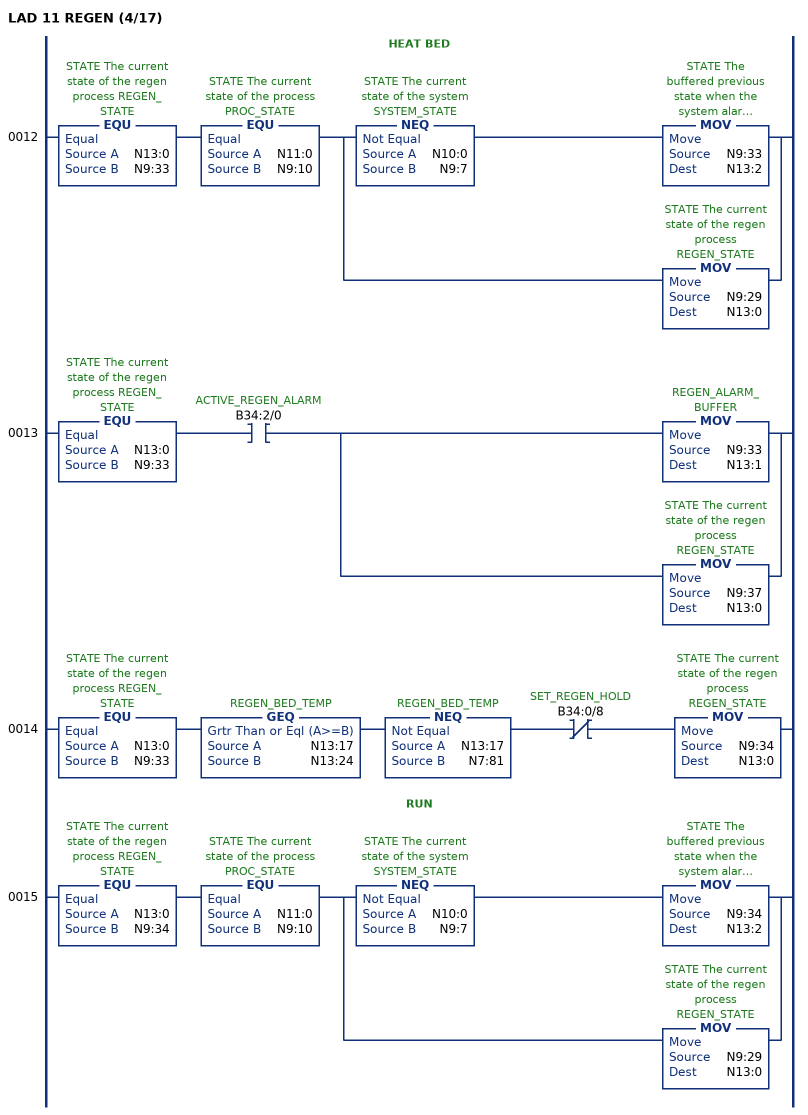
% Rung: 12 %
% TITLE: HEAT BED %
SOR EQU N13:0 N9:33 EQU N11:0 N9:10 BST NEQ N10:0 N9:7 MOV N9:33 N13:2 NXB MOV N9:29 N13:0 BND EOR
%   N13:0  REGEN_STATE  "STATE The current state of the regen process" %
%   N9:33  REGEN_HEAT_BED  "STATE Regen Heat wall" %
%   N11:0  PROC_STATE  "STATE The current state of the process" %
%   N9:10  PROC_STANDBY  "STATE Process Standby" %
%   N10:0  SYSTEM_STATE  "STATE The current state of the system" %
%   N9:7  SYSTEM_COLD_START %
%   N13:2  REGEN_SYSTEM_BUFFER  "STATE The buffered previous state when the system alarm occured" %
%   N9:29  REGEN_IDLE %
% Rung: 13 %
SOR EQU N13:0 N9:33 XIC B34:2/0 BST MOV N9:33 N13:1 NXB MOV N9:37 N13:0 BND EOR
%   N13:0  REGEN_STATE  "STATE The current state of the regen process" %
%   N9:33  REGEN_HEAT_BED  "STATE Regen Heat wall" %
%   B34:2/0  ACTIVE_REGEN_ALARM %
%   N13:1  REGEN_ALARM_BUFFER %
%   N9:37  REGEN_ALARM  "STATE Regen Alarm" %
% Rung: 14 %
SOR EQU N13:0 N9:33 GEQ N13:17 N13:24 NEQ N13:17 N7:81 XIO B34:0/8 MOV N9:34 N13:0 EOR
%   N13:0  REGEN_STATE  "STATE The current state of the regen process" %
%   N9:33  REGEN_HEAT_BED  "STATE Regen Heat wall" %
%   N13:17  REGEN_BED_TEMP %
%   N13:24  ADS_BED_TEMP_HIGH  "CONFIG The temp at which the regen process may continue" %
%   N7:81  TC_OPEN_SP  "CONFIG The value read by an open TC input" %
%   B34:0/8  SET_REGEN_HOLD %
%   N9:34  REGEN_RUN  "STATE Regen Running" %
% Rung: 15 %
% TITLE: RUN %
SOR EQU N13:0 N9:34 EQU N11:0 N9:10 BST NEQ N10:0 N9:7 MOV N9:34 N13:2 NXB MOV N9:29 N13:0 BND EOR
%   N13:0  REGEN_STATE  "STATE The current state of the regen process" %
%   N9:34  REGEN_RUN  "STATE Regen Running" %
%   N11:0  PROC_STATE  "STATE The current state of the process" %
%   N9:10  PROC_STANDBY  "STATE Process Standby" %
%   N10:0  SYSTEM_STATE  "STATE The current state of the system" %
%   N9:7  SYSTEM_COLD_START %
%   N13:2  REGEN_SYSTEM_BUFFER  "STATE The buffered previous state when the system alarm occured" %
%   N9:29  REGEN_IDLE %

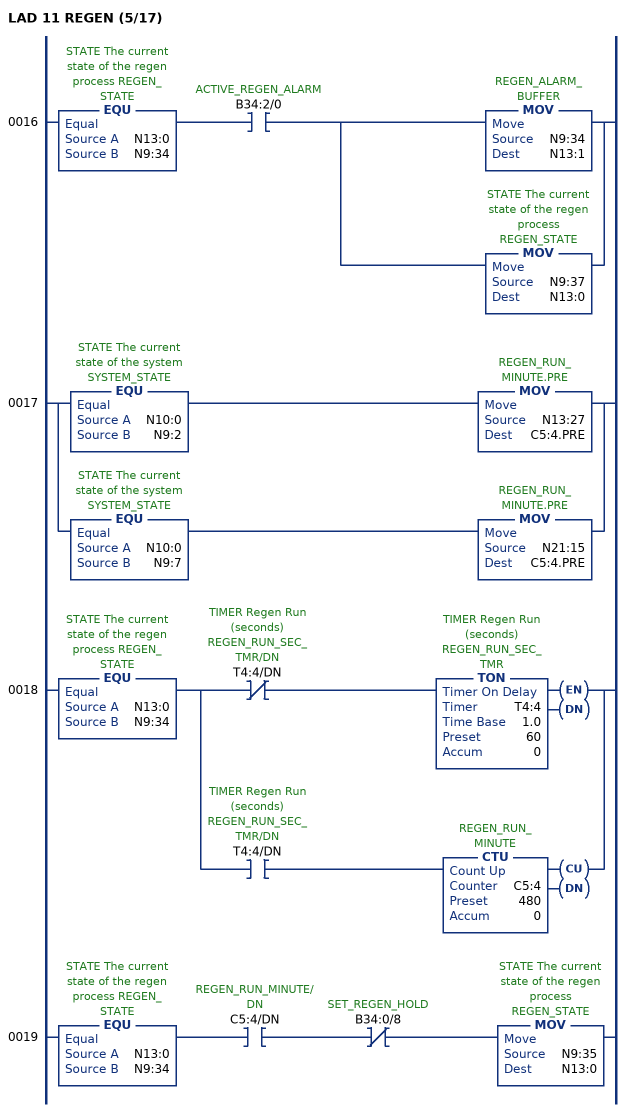
% Rung: 16 %
SOR EQU N13:0 N9:34 XIC B34:2/0 BST MOV N9:34 N13:1 NXB MOV N9:37 N13:0 BND EOR
%   N13:0  REGEN_STATE  "STATE The current state of the regen process" %
%   N9:34  REGEN_RUN  "STATE Regen Running" %
%   B34:2/0  ACTIVE_REGEN_ALARM %
%   N13:1  REGEN_ALARM_BUFFER %
%   N9:37  REGEN_ALARM  "STATE Regen Alarm" %
% Rung: 17 %
SOR BST EQU N10:0 N9:2 MOV N13:27 C5:4.PRE NXB EQU N10:0 N9:7 MOV N21:15 C5:4.PRE BND EOR
%   N10:0  SYSTEM_STATE  "STATE The current state of the system" %
%   N9:2  SYSTEM_PROCESS  "STATE System Process" %
%   N13:27  REGEN_RUN_TIME %
%   C5:4  REGEN_RUN_MINUTE %
%   N9:7  SYSTEM_COLD_START %
%   N21:15  START_REG_RUN_TIME %
% Rung: 18 %
SOR EQU N13:0 N9:34 BST XIO T4:4/DN TON T4:4 1.0 60 0 NXB XIC T4:4/DN CTU C5:4 480 0 BND EOR
%   N13:0  REGEN_STATE  "STATE The current state of the regen process" %
%   N9:34  REGEN_RUN  "STATE Regen Running" %
%   T4:4  REGEN_RUN_SEC_TMR  "TIMER Regen Run (seconds)" %
%   C5:4  REGEN_RUN_MINUTE %
% Rung: 19 %
SOR EQU N13:0 N9:34 XIC C5:4/DN XIO B34:0/8 MOV N9:35 N13:0 EOR
%   N13:0  REGEN_STATE  "STATE The current state of the regen process" %
%   N9:34  REGEN_RUN  "STATE Regen Running" %
%   C5:4  REGEN_RUN_MINUTE %
%   B34:0/8  SET_REGEN_HOLD %
%   N9:35  REGEN_COOL_WALL  "STATE Regen Cool wall" %

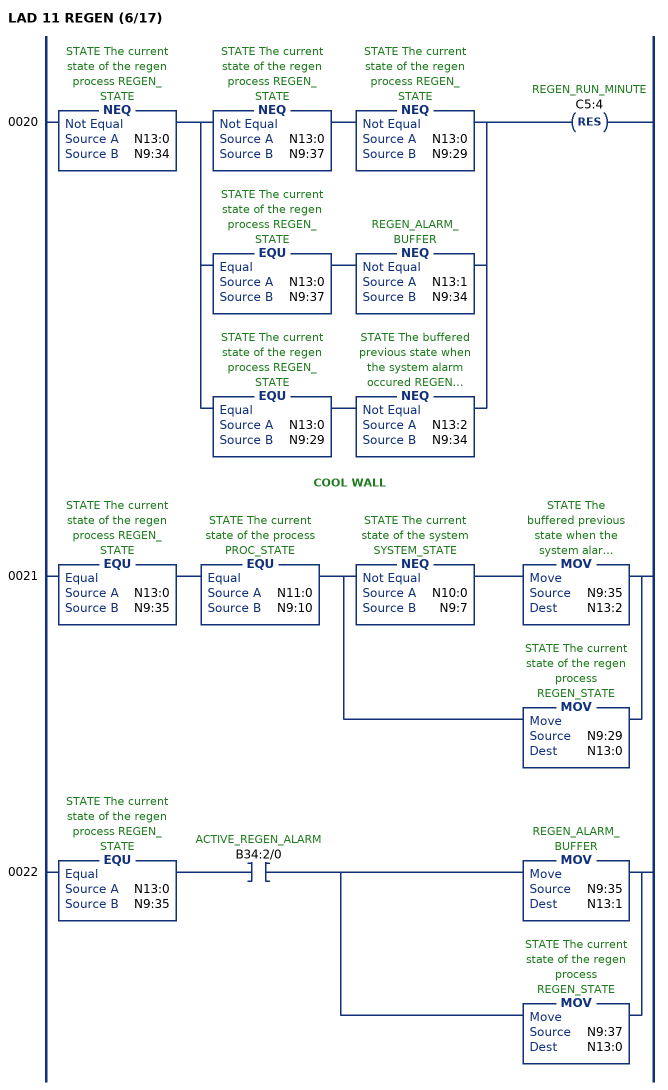
% Rung: 20 %
SOR NEQ N13:0 N9:34 BST NEQ N13:0 N9:37 NEQ N13:0 N9:29 NXB EQU N13:0 N9:37 NEQ N13:1 N9:34 NXB EQU N13:0 N9:29 NEQ N13:2 N9:34 BND RES C5:4 EOR
%   N13:0  REGEN_STATE  "STATE The current state of the regen process" %
%   N9:34  REGEN_RUN  "STATE Regen Running" %
%   N9:37  REGEN_ALARM  "STATE Regen Alarm" %
%   N9:29  REGEN_IDLE %
%   N13:1  REGEN_ALARM_BUFFER %
%   N13:2  REGEN_SYSTEM_BUFFER  "STATE The buffered previous state when the system alarm occured" %
%   C5:4  REGEN_RUN_MINUTE %
% Rung: 21 %
% TITLE: COOL WALL %
SOR EQU N13:0 N9:35 EQU N11:0 N9:10 BST NEQ N10:0 N9:7 MOV N9:35 N13:2 NXB MOV N9:29 N13:0 BND EOR
%   N13:0  REGEN_STATE  "STATE The current state of the regen process" %
%   N9:35  REGEN_COOL_WALL  "STATE Regen Cool wall" %
%   N11:0  PROC_STATE  "STATE The current state of the process" %
%   N9:10  PROC_STANDBY  "STATE Process Standby" %
%   N10:0  SYSTEM_STATE  "STATE The current state of the system" %
%   N9:7  SYSTEM_COLD_START %
%   N13:2  REGEN_SYSTEM_BUFFER  "STATE The buffered previous state when the system alarm occured" %
%   N9:29  REGEN_IDLE %
% Rung: 22 %
SOR EQU N13:0 N9:35 XIC B34:2/0 BST MOV N9:35 N13:1 NXB MOV N9:37 N13:0 BND EOR
%   N13:0  REGEN_STATE  "STATE The current state of the regen process" %
%   N9:35  REGEN_COOL_WALL  "STATE Regen Cool wall" %
%   B34:2/0  ACTIVE_REGEN_ALARM %
%   N13:1  REGEN_ALARM_BUFFER %
%   N9:37  REGEN_ALARM  "STATE Regen Alarm" %

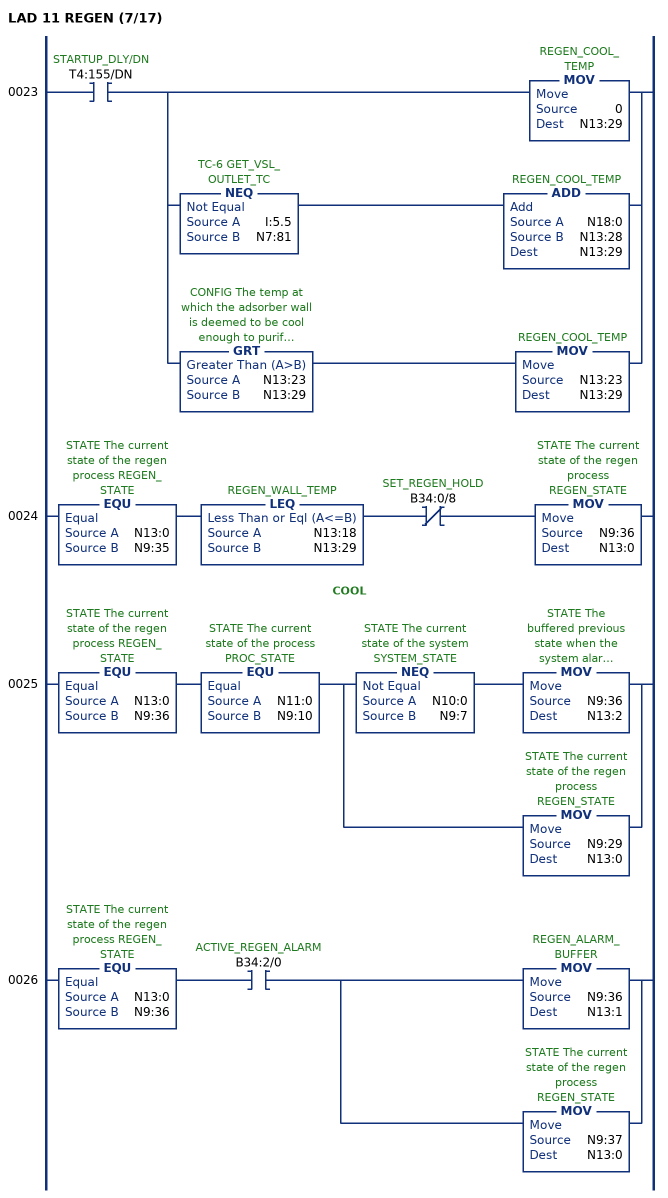
% Rung: 23 %
SOR XIC T4:155/DN BST MOV 0 N13:29 NXB NEQ I:5.5 N7:81 ADD N18:0 N13:28 N13:29 NXB GRT N13:23 N13:29 MOV N13:23 N13:29 BND EOR
%   T4:155  STARTUP_DLY %
%   N13:29  REGEN_COOL_TEMP %
%   I:5.5  GET_VSL_OUTLET_TC  "TC-6" %
%   N7:81  TC_OPEN_SP  "CONFIG The value read by an open TC input" %
%   N18:0  GET_VSL_OUT_GAS_TEMP %
%   N13:28  REGEN_COOL_DIFF %
%   N13:23  ADS_WALL_TEMP_COOL  "CONFIG The temp at which the adsorber wall is deemed to be cool enough to purify" %
% Rung: 24 %
SOR EQU N13:0 N9:35 LEQ N13:18 N13:29 XIO B34:0/8 MOV N9:36 N13:0 EOR
%   N13:0  REGEN_STATE  "STATE The current state of the regen process" %
%   N9:35  REGEN_COOL_WALL  "STATE Regen Cool wall" %
%   N13:18  REGEN_WALL_TEMP %
%   N13:29  REGEN_COOL_TEMP %
%   B34:0/8  SET_REGEN_HOLD %
%   N9:36  REGEN_COOL  "STATE Regen Cool" %
% Rung: 25 %
% TITLE: COOL %
SOR EQU N13:0 N9:36 EQU N11:0 N9:10 BST NEQ N10:0 N9:7 MOV N9:36 N13:2 NXB MOV N9:29 N13:0 BND EOR
%   N13:0  REGEN_STATE  "STATE The current state of the regen process" %
%   N9:36  REGEN_COOL  "STATE Regen Cool" %
%   N11:0  PROC_STATE  "STATE The current state of the process" %
%   N9:10  PROC_STANDBY  "STATE Process Standby" %
%   N10:0  SYSTEM_STATE  "STATE The current state of the system" %
%   N9:7  SYSTEM_COLD_START %
%   N13:2  REGEN_SYSTEM_BUFFER  "STATE The buffered previous state when the system alarm occured" %
%   N9:29  REGEN_IDLE %
% Rung: 26 %
SOR EQU N13:0 N9:36 XIC B34:2/0 BST MOV N9:36 N13:1 NXB MOV N9:37 N13:0 BND EOR
%   N13:0  REGEN_STATE  "STATE The current state of the regen process" %
%   N9:36  REGEN_COOL  "STATE Regen Cool" %
%   B34:2/0  ACTIVE_REGEN_ALARM %
%   N13:1  REGEN_ALARM_BUFFER %
%   N9:37  REGEN_ALARM  "STATE Regen Alarm" %

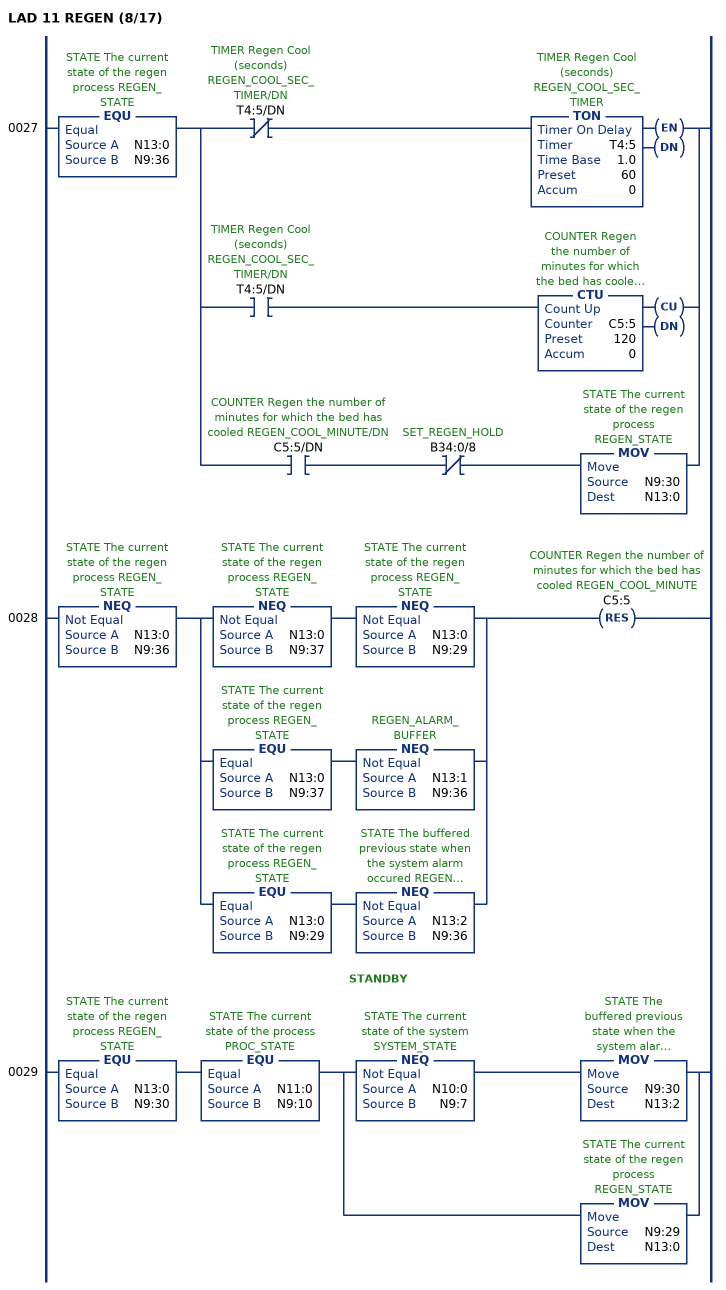
% Rung: 27 %
SOR EQU N13:0 N9:36 BST XIO T4:5/DN TON T4:5 1.0 60 0 NXB XIC T4:5/DN CTU C5:5 120 0 NXB XIC C5:5/DN XIO B34:0/8 MOV N9:30 N13:0 BND EOR
%   N13:0  REGEN_STATE  "STATE The current state of the regen process" %
%   N9:36  REGEN_COOL  "STATE Regen Cool" %
%   T4:5  REGEN_COOL_SEC_TIMER  "TIMER Regen Cool (seconds)" %
%   C5:5  REGEN_COOL_MINUTE  "COUNTER Regen the number of minutes for which the bed has cooled" %
%   B34:0/8  SET_REGEN_HOLD %
%   N9:30  REGEN_STANDBY  "STATE Regen Standby" %
% Rung: 28 %
SOR NEQ N13:0 N9:36 BST NEQ N13:0 N9:37 NEQ N13:0 N9:29 NXB EQU N13:0 N9:37 NEQ N13:1 N9:36 NXB EQU N13:0 N9:29 NEQ N13:2 N9:36 BND RES C5:5 EOR
%   N13:0  REGEN_STATE  "STATE The current state of the regen process" %
%   N9:36  REGEN_COOL  "STATE Regen Cool" %
%   N9:37  REGEN_ALARM  "STATE Regen Alarm" %
%   N9:29  REGEN_IDLE %
%   N13:1  REGEN_ALARM_BUFFER %
%   N13:2  REGEN_SYSTEM_BUFFER  "STATE The buffered previous state when the system alarm occured" %
%   C5:5  REGEN_COOL_MINUTE  "COUNTER Regen the number of minutes for which the bed has cooled" %
% Rung: 29 %
% TITLE: STANDBY %
SOR EQU N13:0 N9:30 EQU N11:0 N9:10 BST NEQ N10:0 N9:7 MOV N9:30 N13:2 NXB MOV N9:29 N13:0 BND EOR
%   N13:0  REGEN_STATE  "STATE The current state of the regen process" %
%   N9:30  REGEN_STANDBY  "STATE Regen Standby" %
%   N11:0  PROC_STATE  "STATE The current state of the process" %
%   N9:10  PROC_STANDBY  "STATE Process Standby" %
%   N10:0  SYSTEM_STATE  "STATE The current state of the system" %
%   N9:7  SYSTEM_COLD_START %
%   N13:2  REGEN_SYSTEM_BUFFER  "STATE The buffered previous state when the system alarm occured" %
%   N9:29  REGEN_IDLE %

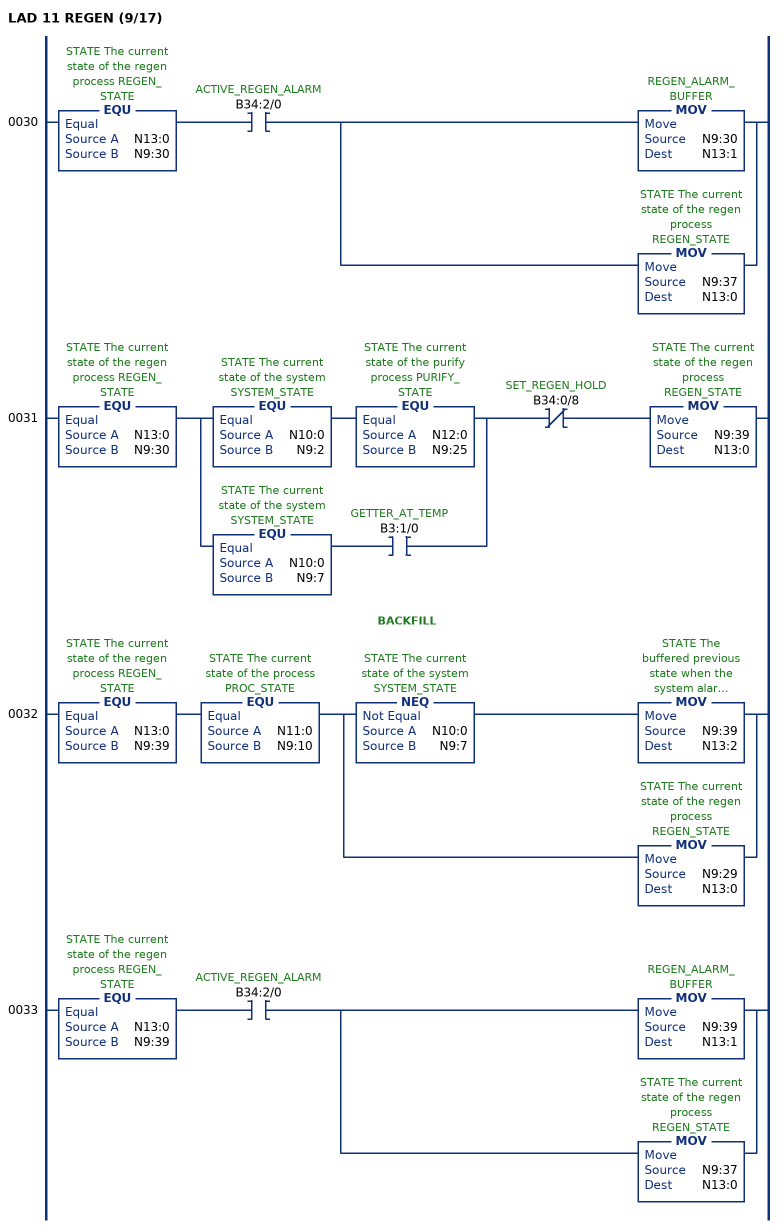
% Rung: 30 %
SOR EQU N13:0 N9:30 XIC B34:2/0 BST MOV N9:30 N13:1 NXB MOV N9:37 N13:0 BND EOR
%   N13:0  REGEN_STATE  "STATE The current state of the regen process" %
%   N9:30  REGEN_STANDBY  "STATE Regen Standby" %
%   B34:2/0  ACTIVE_REGEN_ALARM %
%   N13:1  REGEN_ALARM_BUFFER %
%   N9:37  REGEN_ALARM  "STATE Regen Alarm" %
% Rung: 31 %
SOR EQU N13:0 N9:30 BST EQU N10:0 N9:2 EQU N12:0 N9:25 NXB EQU N10:0 N9:7 XIC B3:1/0 BND XIO B34:0/8 MOV N9:39 N13:0 EOR
%   N13:0  REGEN_STATE  "STATE The current state of the regen process" %
%   N9:30  REGEN_STANDBY  "STATE Regen Standby" %
%   N10:0  SYSTEM_STATE  "STATE The current state of the system" %
%   N9:2  SYSTEM_PROCESS  "STATE System Process" %
%   N12:0  PURIFY_STATE  "STATE The current state of the purify process" %
%   N9:25  PURIFY_DONE %
%   N9:7  SYSTEM_COLD_START %
%   B3:1/0  GETTER_AT_TEMP %
%   B34:0/8  SET_REGEN_HOLD %
%   N9:39  REGEN_BACKFILL %
% Rung: 32 %
% TITLE: BACKFILL %
SOR EQU N13:0 N9:39 EQU N11:0 N9:10 BST NEQ N10:0 N9:7 MOV N9:39 N13:2 NXB MOV N9:29 N13:0 BND EOR
%   N13:0  REGEN_STATE  "STATE The current state of the regen process" %
%   N9:39  REGEN_BACKFILL %
%   N11:0  PROC_STATE  "STATE The current state of the process" %
%   N9:10  PROC_STANDBY  "STATE Process Standby" %
%   N10:0  SYSTEM_STATE  "STATE The current state of the system" %
%   N9:7  SYSTEM_COLD_START %
%   N13:2  REGEN_SYSTEM_BUFFER  "STATE The buffered previous state when the system alarm occured" %
%   N9:29  REGEN_IDLE %
% Rung: 33 %
SOR EQU N13:0 N9:39 XIC B34:2/0 BST MOV N9:39 N13:1 NXB MOV N9:37 N13:0 BND EOR
%   N13:0  REGEN_STATE  "STATE The current state of the regen process" %
%   N9:39  REGEN_BACKFILL %
%   B34:2/0  ACTIVE_REGEN_ALARM %
%   N13:1  REGEN_ALARM_BUFFER %
%   N9:37  REGEN_ALARM  "STATE Regen Alarm" %

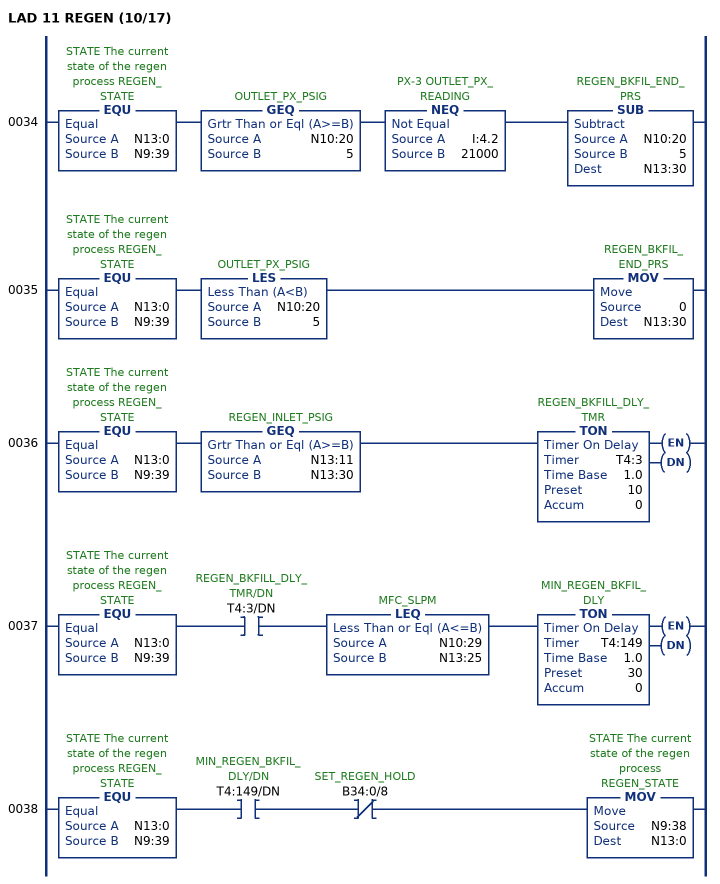
% Rung: 34 %
SOR EQU N13:0 N9:39 GEQ N10:20 5 NEQ I:4.2 21000 SUB N10:20 5 N13:30 EOR
%   N13:0  REGEN_STATE  "STATE The current state of the regen process" %
%   N9:39  REGEN_BACKFILL %
%   N10:20  OUTLET_PX_PSIG %
%   I:4.2  OUTLET_PX_READING  "PX-3" %
%   N13:30  REGEN_BKFIL_END_PRS %
% Rung: 35 %
SOR EQU N13:0 N9:39 LES N10:20 5 MOV 0 N13:30 EOR
%   N13:0  REGEN_STATE  "STATE The current state of the regen process" %
%   N9:39  REGEN_BACKFILL %
%   N10:20  OUTLET_PX_PSIG %
%   N13:30  REGEN_BKFIL_END_PRS %
% Rung: 36 %
SOR EQU N13:0 N9:39 GEQ N13:11 N13:30 TON T4:3 1.0 10 0 EOR
%   N13:0  REGEN_STATE  "STATE The current state of the regen process" %
%   N9:39  REGEN_BACKFILL %
%   N13:11  REGEN_INLET_PSIG %
%   N13:30  REGEN_BKFIL_END_PRS %
%   T4:3  REGEN_BKFILL_DLY_TMR %
% Rung: 37 %
SOR EQU N13:0 N9:39 XIC T4:3/DN LEQ N10:29 N13:25 TON T4:149 1.0 30 0 EOR
%   N13:0  REGEN_STATE  "STATE The current state of the regen process" %
%   N9:39  REGEN_BACKFILL %
%   T4:3  REGEN_BKFILL_DLY_TMR %
%   N10:29  MFC_SLPM %
%   N13:25  REGEN_BKFIL_END_FLOW %
%   T4:149  MIN_REGEN_BKFIL_DLY %
% Rung: 38 %
SOR EQU N13:0 N9:39 XIC T4:149/DN XIO B34:0/8 MOV N9:38 N13:0 EOR
%   N13:0  REGEN_STATE  "STATE The current state of the regen process" %
%   N9:39  REGEN_BACKFILL %
%   T4:149  MIN_REGEN_BKFIL_DLY %
%   B34:0/8  SET_REGEN_HOLD %
%   N9:38  REGEN_DONE %

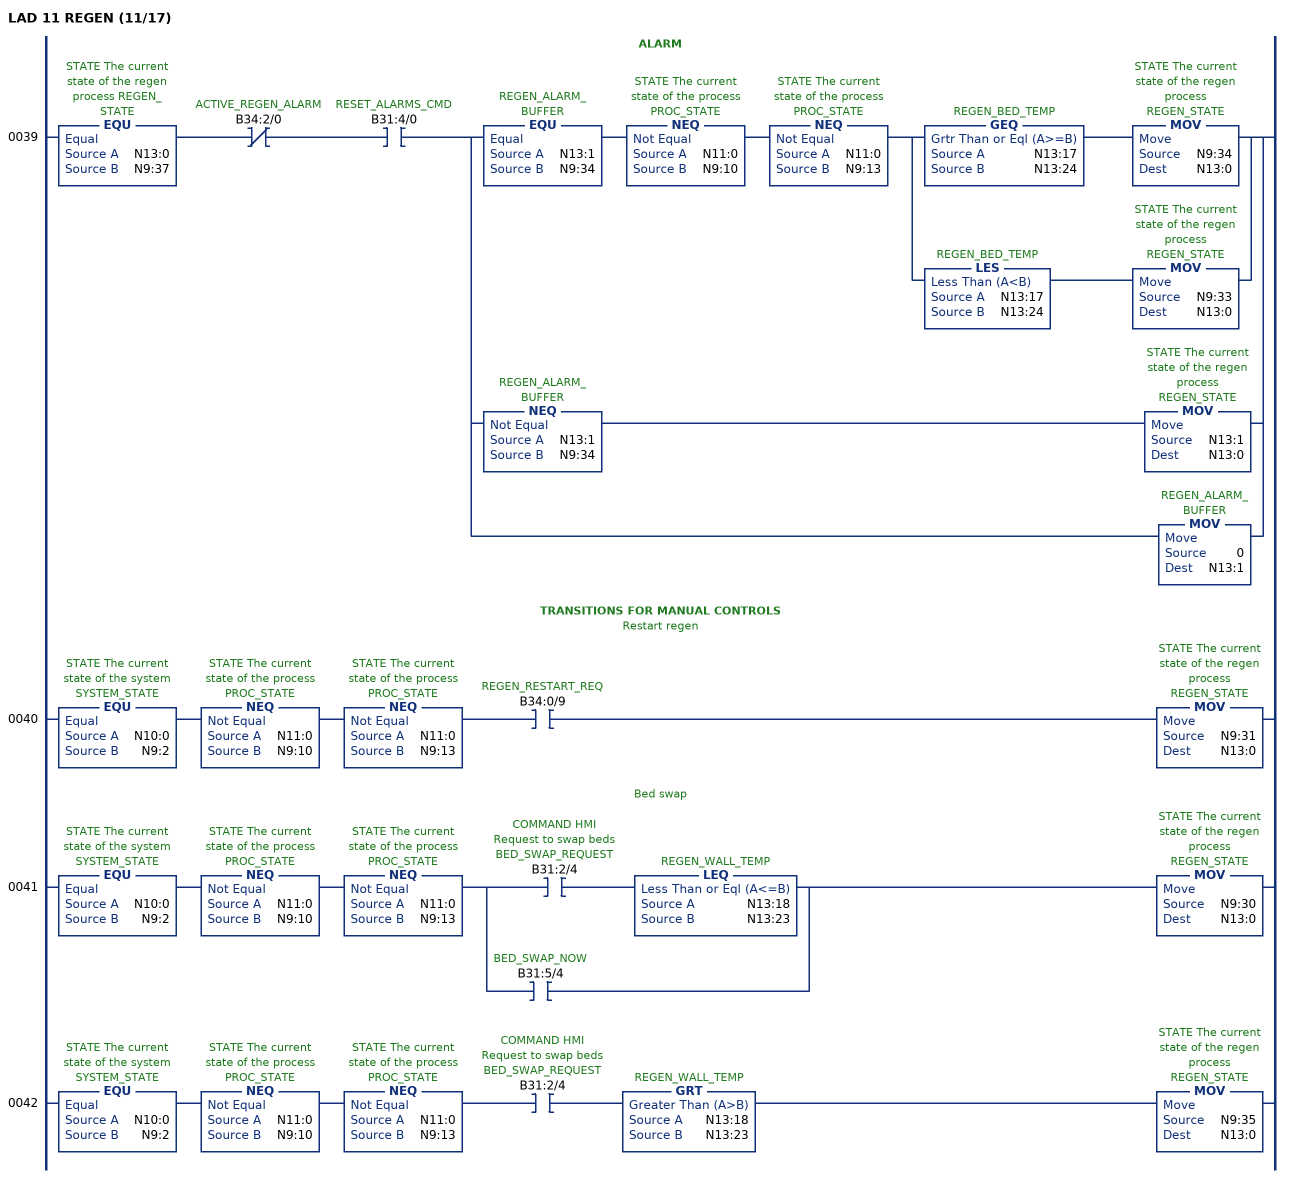
% Rung: 39 %
% TITLE: ALARM %
SOR EQU N13:0 N9:37 XIO B34:2/0 XIC B31:4/0 BST EQU N13:1 N9:34 NEQ N11:0 N9:10 NEQ N11:0 N9:13 BST GEQ N13:17 N13:24 MOV N9:34 N13:0 NXB LES N13:17 N13:24 MOV N9:33 N13:0 BND NXB NEQ N13:1 N9:34 MOV N13:1 N13:0 NXB MOV 0 N13:1 BND EOR
%   N13:0  REGEN_STATE  "STATE The current state of the regen process" %
%   N9:37  REGEN_ALARM  "STATE Regen Alarm" %
%   B34:2/0  ACTIVE_REGEN_ALARM %
%   B31:4/0  RESET_ALARMS_CMD %
%   N13:1  REGEN_ALARM_BUFFER %
%   N9:34  REGEN_RUN  "STATE Regen Running" %
%   N11:0  PROC_STATE  "STATE The current state of the process" %
%   N9:10  PROC_STANDBY  "STATE Process Standby" %
%   N9:13  PROC_OVERLAP  "STATE Process Purify Overlap" %
%   N13:17  REGEN_BED_TEMP %
%   N13:24  ADS_BED_TEMP_HIGH  "CONFIG The temp at which the regen process may continue" %
%   N9:33  REGEN_HEAT_BED  "STATE Regen Heat wall" %
% Rung: 40 %
% TITLE: TRANSITIONS FOR MANUAL CONTROLS %
% Restart regen %
SOR EQU N10:0 N9:2 NEQ N11:0 N9:10 NEQ N11:0 N9:13 XIC B34:0/9 MOV N9:31 N13:0 EOR
%   N10:0  SYSTEM_STATE  "STATE The current state of the system" %
%   N9:2  SYSTEM_PROCESS  "STATE System Process" %
%   N11:0  PROC_STATE  "STATE The current state of the process" %
%   N9:10  PROC_STANDBY  "STATE Process Standby" %
%   N9:13  PROC_OVERLAP  "STATE Process Purify Overlap" %
%   B34:0/9  REGEN_RESTART_REQ %
%   N9:31  REGEN_DELAY  "STATE Regen Delay" %
%   N13:0  REGEN_STATE  "STATE The current state of the regen process" %
% Rung: 41 %
% Bed swap %
SOR EQU N10:0 N9:2 NEQ N11:0 N9:10 NEQ N11:0 N9:13 BST XIC B31:2/4 LEQ N13:18 N13:23 NXB XIC B31:5/4 BND MOV N9:30 N13:0 EOR
%   N10:0  SYSTEM_STATE  "STATE The current state of the system" %
%   N9:2  SYSTEM_PROCESS  "STATE System Process" %
%   N11:0  PROC_STATE  "STATE The current state of the process" %
%   N9:10  PROC_STANDBY  "STATE Process Standby" %
%   N9:13  PROC_OVERLAP  "STATE Process Purify Overlap" %
%   B31:2/4  BED_SWAP_REQUEST  "COMMAND HMI Request to swap beds" %
%   N13:18  REGEN_WALL_TEMP %
%   N13:23  ADS_WALL_TEMP_COOL  "CONFIG The temp at which the adsorber wall is deemed to be cool enough to purify" %
%   B31:5/4  BED_SWAP_NOW %
%   N9:30  REGEN_STANDBY  "STATE Regen Standby" %
%   N13:0  REGEN_STATE  "STATE The current state of the regen process" %
% Rung: 42 %
SOR EQU N10:0 N9:2 NEQ N11:0 N9:10 NEQ N11:0 N9:13 XIC B31:2/4 GRT N13:18 N13:23 MOV N9:35 N13:0 EOR
%   N10:0  SYSTEM_STATE  "STATE The current state of the system" %
%   N9:2  SYSTEM_PROCESS  "STATE System Process" %
%   N11:0  PROC_STATE  "STATE The current state of the process" %
%   N9:10  PROC_STANDBY  "STATE Process Standby" %
%   N9:13  PROC_OVERLAP  "STATE Process Purify Overlap" %
%   B31:2/4  BED_SWAP_REQUEST  "COMMAND HMI Request to swap beds" %
%   N13:18  REGEN_WALL_TEMP %
%   N13:23  ADS_WALL_TEMP_COOL  "CONFIG The temp at which the adsorber wall is deemed to be cool enough to purify" %
%   N9:35  REGEN_COOL_WALL  "STATE Regen Cool wall" %
%   N13:0  REGEN_STATE  "STATE The current state of the regen process" %

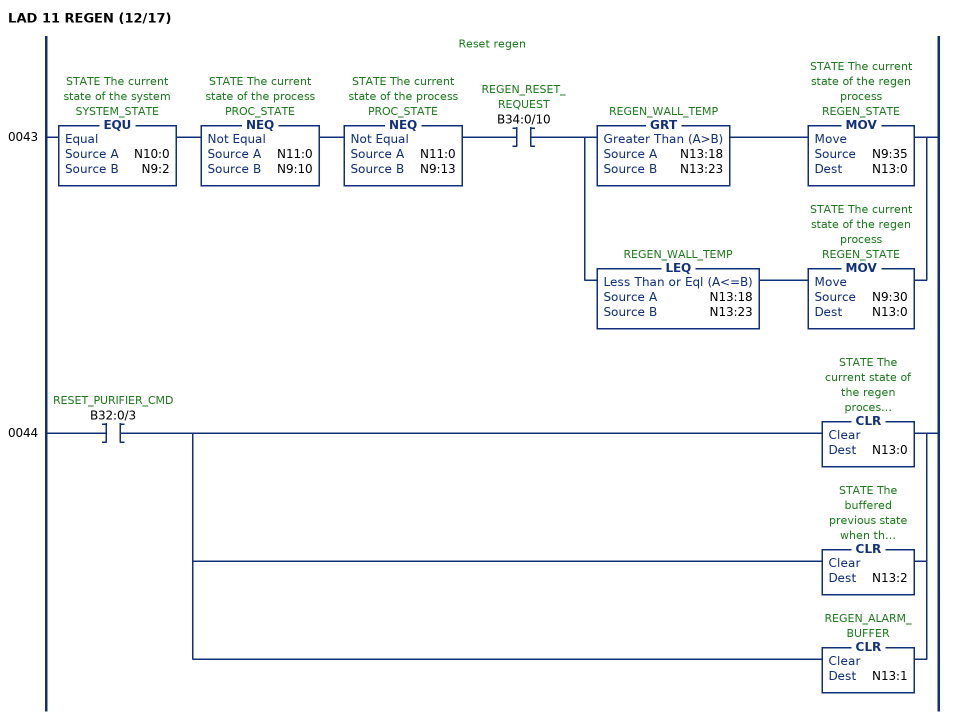
% Rung: 43 %
% Reset regen %
SOR EQU N10:0 N9:2 NEQ N11:0 N9:10 NEQ N11:0 N9:13 XIC B34:0/10 BST GRT N13:18 N13:23 MOV N9:35 N13:0 NXB LEQ N13:18 N13:23 MOV N9:30 N13:0 BND EOR
%   N10:0  SYSTEM_STATE  "STATE The current state of the system" %
%   N9:2  SYSTEM_PROCESS  "STATE System Process" %
%   N11:0  PROC_STATE  "STATE The current state of the process" %
%   N9:10  PROC_STANDBY  "STATE Process Standby" %
%   N9:13  PROC_OVERLAP  "STATE Process Purify Overlap" %
%   B34:0/10  REGEN_RESET_REQUEST %
%   N13:18  REGEN_WALL_TEMP %
%   N13:23  ADS_WALL_TEMP_COOL  "CONFIG The temp at which the adsorber wall is deemed to be cool enough to purify" %
%   N9:35  REGEN_COOL_WALL  "STATE Regen Cool wall" %
%   N13:0  REGEN_STATE  "STATE The current state of the regen process" %
%   N9:30  REGEN_STANDBY  "STATE Regen Standby" %
% Rung: 44 %
SOR XIC B32:0/3 BST CLR N13:0 NXB CLR N13:2 NXB CLR N13:1 BND EOR
%   B32:0/3  RESET_PURIFIER_CMD %
%   N13:0  REGEN_STATE  "STATE The current state of the regen process" %
%   N13:2  REGEN_SYSTEM_BUFFER  "STATE The buffered previous state when the system alarm occured" %
%   N13:1  REGEN_ALARM_BUFFER %

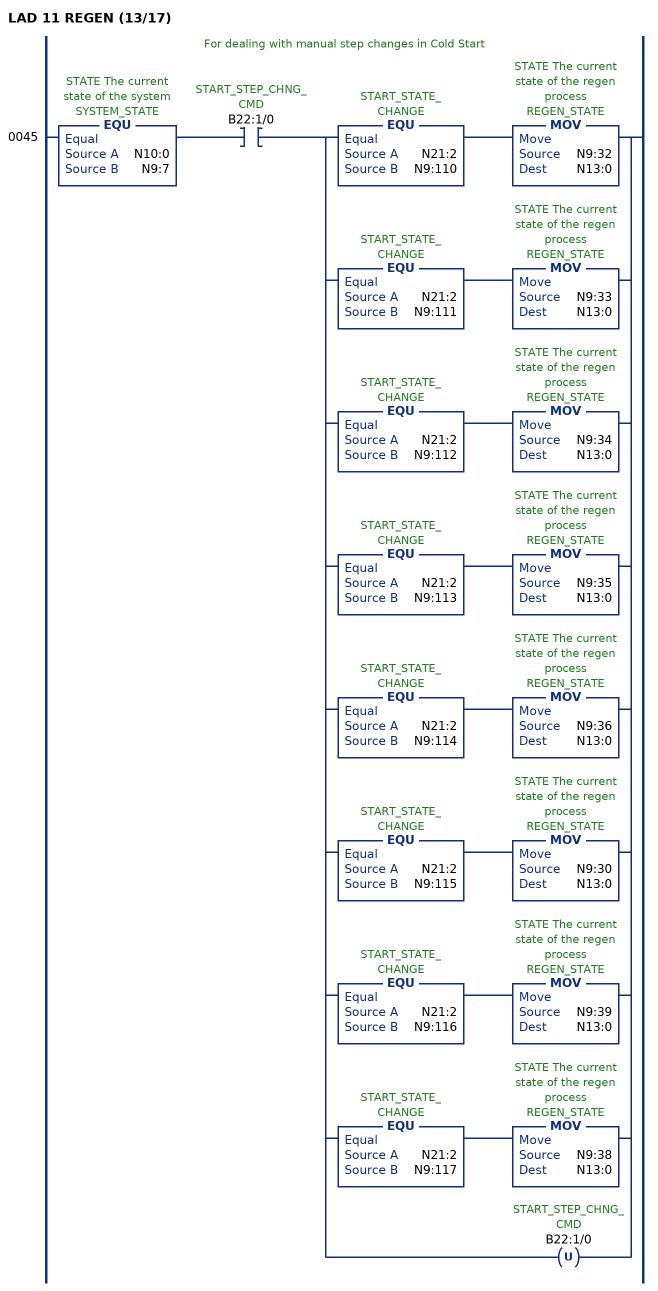
% Rung: 45 %
% For dealing with manual step changes in Cold Start %
SOR EQU N10:0 N9:7 XIC B22:1/0 BST EQU N21:2 N9:110 MOV N9:32 N13:0 NXB EQU N21:2 N9:111 MOV N9:33 N13:0 NXB EQU N21:2 N9:112 MOV N9:34 N13:0 NXB EQU N21:2 N9:113 MOV N9:35 N13:0 NXB EQU N21:2 N9:114 MOV N9:36 N13:0 NXB EQU N21:2 N9:115 MOV N9:30 N13:0 NXB EQU N21:2 N9:116 MOV N9:39 N13:0 NXB EQU N21:2 N9:117 MOV N9:38 N13:0 NXB OTU B22:1/0 BND EOR
%   N10:0  SYSTEM_STATE  "STATE The current state of the system" %
%   N9:7  SYSTEM_COLD_START %
%   B22:1/0  START_STEP_CHNG_CMD %
%   N21:2  START_STATE_CHANGE %
%   N9:110  START_REG_VENT %
%   N9:32  REGEN_VENT  "STATE Regen Vent" %
%   N13:0  REGEN_STATE  "STATE The current state of the regen process" %
%   N9:111  START_REG_HEAT %
%   N9:33  REGEN_HEAT_BED  "STATE Regen Heat wall" %
%   N9:112  START_REG_RUN %
%   N9:34  REGEN_RUN  "STATE Regen Running" %
%   N9:113  START_REG_COOL %
%   N9:35  REGEN_COOL_WALL  "STATE Regen Cool wall" %
%   N9:114  START_REG_TIMED_COOL %
%   N9:36  REGEN_COOL  "STATE Regen Cool" %
%   N9:115  START_REG_STANDBY %
%   N9:30  REGEN_STANDBY  "STATE Regen Standby" %
%   N9:116  START_REG_BACKFILL %
%   N9:39  REGEN_BACKFILL %
%   N9:117  START_REG_DONE %
%   N9:38  REGEN_DONE %

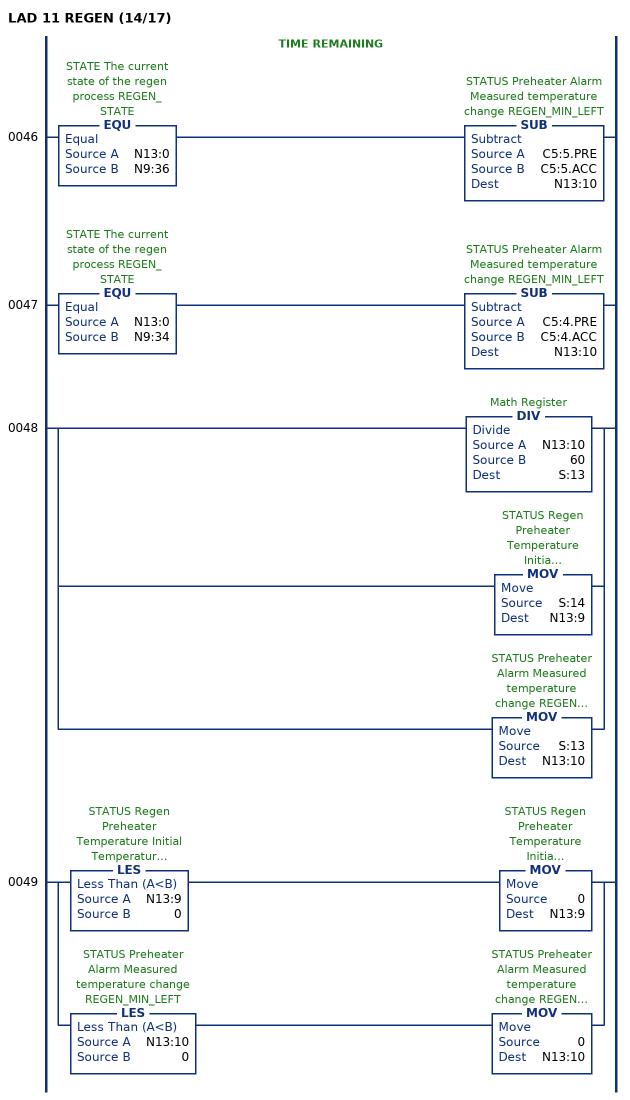
% Rung: 46 %
% TITLE: TIME REMAINING %
SOR EQU N13:0 N9:36 SUB C5:5.PRE C5:5.ACC N13:10 EOR
%   N13:0  REGEN_STATE  "STATE The current state of the regen process" %
%   N9:36  REGEN_COOL  "STATE Regen Cool" %
%   C5:5  REGEN_COOL_MINUTE  "COUNTER Regen the number of minutes for which the bed has cooled" %
%   N13:10  REGEN_MIN_LEFT  "STATUS Preheater Alarm Measured temperature change" %
% Rung: 47 %
SOR EQU N13:0 N9:34 SUB C5:4.PRE C5:4.ACC N13:10 EOR
%   N13:0  REGEN_STATE  "STATE The current state of the regen process" %
%   N9:34  REGEN_RUN  "STATE Regen Running" %
%   C5:4  REGEN_RUN_MINUTE %
%   N13:10  REGEN_MIN_LEFT  "STATUS Preheater Alarm Measured temperature change" %
% Rung: 48 %
SOR BST DIV N13:10 60 S:13 NXB MOV S:14 N13:9 NXB MOV S:13 N13:10 BND EOR
%   N13:10  REGEN_MIN_LEFT  "STATUS Preheater Alarm Measured temperature change" %
%   S:13  "Math Register" %
%   S:14  "Math Register" %
%   N13:9  REGEN_HRS_LEFT  "STATUS Regen Preheater Temperature Initial Temperature" %
% Rung: 49 %
SOR BST LES N13:9 0 MOV 0 N13:9 NXB LES N13:10 0 MOV 0 N13:10 BND EOR
%   N13:9  REGEN_HRS_LEFT  "STATUS Regen Preheater Temperature Initial Temperature" %
%   N13:10  REGEN_MIN_LEFT  "STATUS Preheater Alarm Measured temperature change" %

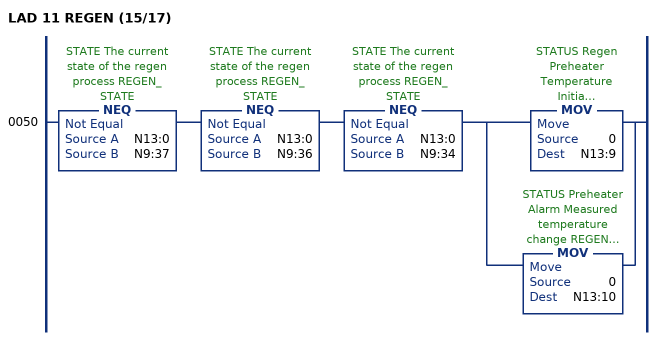
% Rung: 50 %
SOR NEQ N13:0 N9:37 NEQ N13:0 N9:36 NEQ N13:0 N9:34 BST MOV 0 N13:9 NXB MOV 0 N13:10 BND EOR
%   N13:0  REGEN_STATE  "STATE The current state of the regen process" %
%   N9:37  REGEN_ALARM  "STATE Regen Alarm" %
%   N9:36  REGEN_COOL  "STATE Regen Cool" %
%   N9:34  REGEN_RUN  "STATE Regen Running" %
%   N13:9  REGEN_HRS_LEFT  "STATUS Regen Preheater Temperature Initial Temperature" %
%   N13:10  REGEN_MIN_LEFT  "STATUS Preheater Alarm Measured temperature change" %

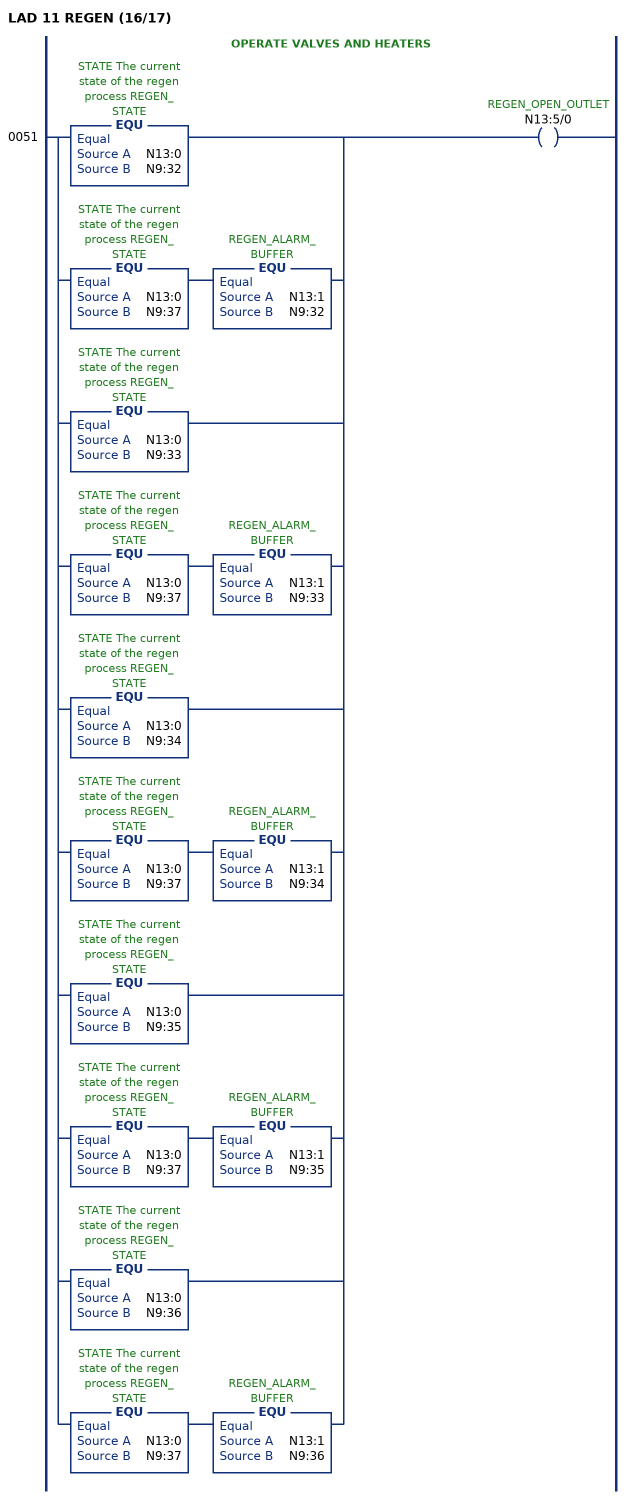
% Rung: 51 %
% TITLE: OPERATE VALVES AND HEATERS %
SOR BST EQU N13:0 N9:32 NXB EQU N13:0 N9:37 EQU N13:1 N9:32 NXB EQU N13:0 N9:33 NXB EQU N13:0 N9:37 EQU N13:1 N9:33 NXB EQU N13:0 N9:34 NXB EQU N13:0 N9:37 EQU N13:1 N9:34 NXB EQU N13:0 N9:35 NXB EQU N13:0 N9:37 EQU N13:1 N9:35 NXB EQU N13:0 N9:36 NXB EQU N13:0 N9:37 EQU N13:1 N9:36 BND OTE N13:5/0 EOR
%   N13:0  REGEN_STATE  "STATE The current state of the regen process" %
%   N9:32  REGEN_VENT  "STATE Regen Vent" %
%   N9:37  REGEN_ALARM  "STATE Regen Alarm" %
%   N13:1  REGEN_ALARM_BUFFER %
%   N9:33  REGEN_HEAT_BED  "STATE Regen Heat wall" %
%   N9:34  REGEN_RUN  "STATE Regen Running" %
%   N9:35  REGEN_COOL_WALL  "STATE Regen Cool wall" %
%   N9:36  REGEN_COOL  "STATE Regen Cool" %
%   N13:5/0  REGEN_OPEN_OUTLET %

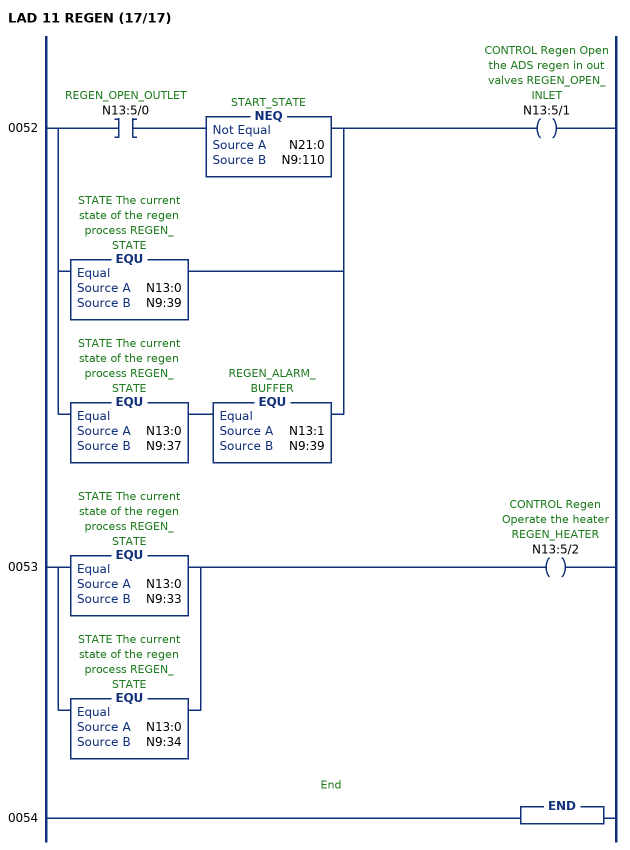
% Rung: 52 %
SOR BST XIC N13:5/0 NEQ N21:0 N9:110 NXB EQU N13:0 N9:39 NXB EQU N13:0 N9:37 EQU N13:1 N9:39 BND OTE N13:5/1 EOR
%   N13:5/0  REGEN_OPEN_OUTLET %
%   N21:0  START_STATE %
%   N9:110  START_REG_VENT %
%   N13:0  REGEN_STATE  "STATE The current state of the regen process" %
%   N9:39  REGEN_BACKFILL %
%   N9:37  REGEN_ALARM  "STATE Regen Alarm" %
%   N13:1  REGEN_ALARM_BUFFER %
%   N13:5/1  REGEN_OPEN_INLET  "CONTROL Regen Open the ADS regen in out valves" %
% Rung: 53 %
SOR BST EQU N13:0 N9:33 NXB EQU N13:0 N9:34 BND OTE N13:5/2 EOR
%   N13:0  REGEN_STATE  "STATE The current state of the regen process" %
%   N9:33  REGEN_HEAT_BED  "STATE Regen Heat wall" %
%   N9:34  REGEN_RUN  "STATE Regen Running" %
%   N13:5/2  REGEN_HEATER  "CONTROL Regen Operate the heater" %
% Rung: 54 %
% End %
SOR END EOR

LADDER 12 "REGEN_FLT"    % regen alarms and warnings %
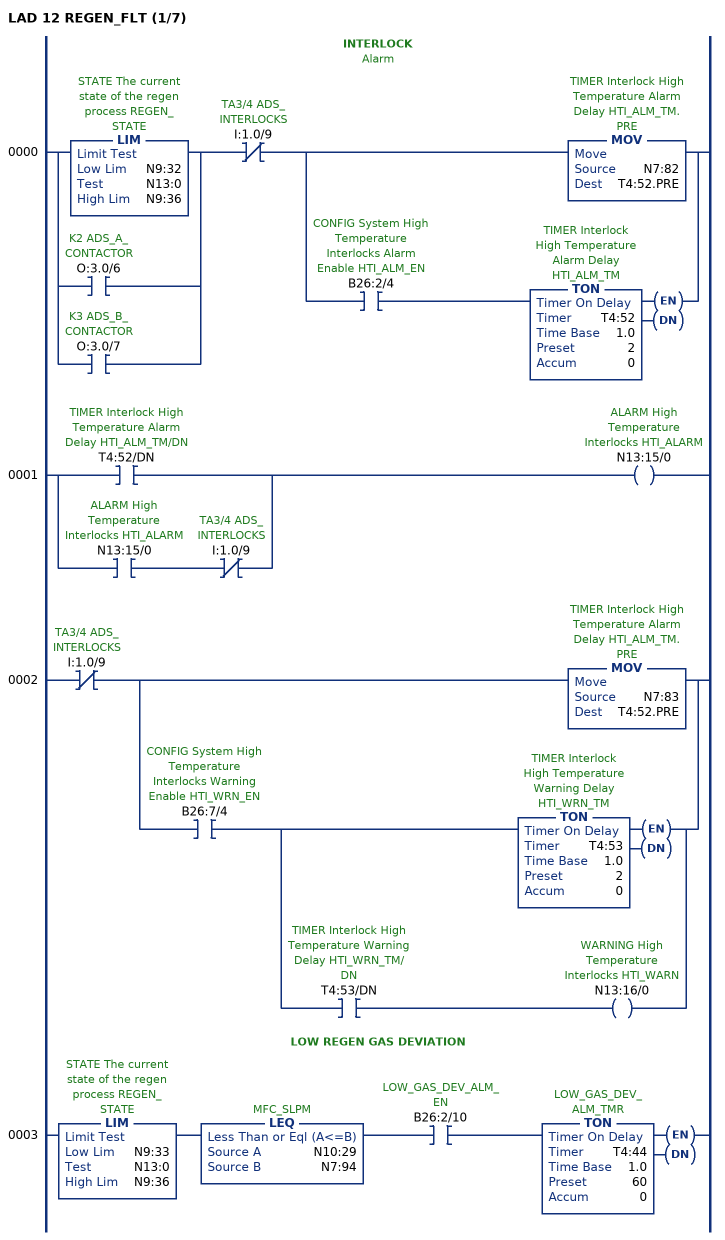
% Rung: 0 %
% TITLE: INTERLOCK %
% Alarm %
SOR BST LIM N9:32 N13:0 N9:36 NXB XIC O:3.0/6 NXB XIC O:3.0/7 BND XIO I:1.0/9 BST MOV N7:82 T4:52.PRE NXB XIC B26:2/4 TON T4:52 1.0 2 0 BND EOR
%   N9:32  REGEN_VENT  "STATE Regen Vent" %
%   N13:0  REGEN_STATE  "STATE The current state of the regen process" %
%   N9:36  REGEN_COOL  "STATE Regen Cool" %
%   O:3.0/6  ADS_A_CONTACTOR  "K2" %
%   O:3.0/7  ADS_B_CONTACTOR  "K3" %
%   I:1.0/9  ADS_INTERLOCKS  "TA3/4" %
%   N7:82  HTI_ALM_DY  "CONFIG Interlocks High Temp Alarm Delay" %
%   T4:52  HTI_ALM_TM  "TIMER Interlock High Temperature Alarm Delay" %
%   B26:2/4  HTI_ALM_EN  "CONFIG System High Temperature Interlocks Alarm Enable" %
% Rung: 1 %
SOR BST XIC T4:52/DN NXB XIC N13:15/0 XIO I:1.0/9 BND OTE N13:15/0 EOR
%   T4:52  HTI_ALM_TM  "TIMER Interlock High Temperature Alarm Delay" %
%   N13:15/0  HTI_ALARM  "ALARM High Temperature Interlocks" %
%   I:1.0/9  ADS_INTERLOCKS  "TA3/4" %
% Rung: 2 %
SOR XIO I:1.0/9 BST MOV N7:83 T4:52.PRE NXB XIC B26:7/4 BST TON T4:53 1.0 2 0 NXB XIC T4:53/DN OTE N13:16/0 BND BND EOR
%   I:1.0/9  ADS_INTERLOCKS  "TA3/4" %
%   N7:83  HTI_WRN_DY  "CONFIG Interlocks High Temp Warning Delay" %
%   T4:52  HTI_ALM_TM  "TIMER Interlock High Temperature Alarm Delay" %
%   B26:7/4  HTI_WRN_EN  "CONFIG System High Temperature Interlocks Warning Enable" %
%   T4:53  HTI_WRN_TM  "TIMER Interlock High Temperature Warning Delay" %
%   N13:16/0  HTI_WARN  "WARNING High Temperature Interlocks" %
% Rung: 3 %
% TITLE: LOW REGEN GAS DEVIATION %
SOR LIM N9:33 N13:0 N9:36 LEQ N10:29 N7:94 XIC B26:2/10 TON T4:44 1.0 60 0 EOR
%   N9:33  REGEN_HEAT_BED  "STATE Regen Heat wall" %
%   N13:0  REGEN_STATE  "STATE The current state of the regen process" %
%   N9:36  REGEN_COOL  "STATE Regen Cool" %
%   N10:29  MFC_SLPM %
%   N7:94  LOW_GAS_DEV_ALM_SP %
%   B26:2/10  LOW_GAS_DEV_ALM_EN %
%   T4:44  LOW_GAS_DEV_ALM_TMR %

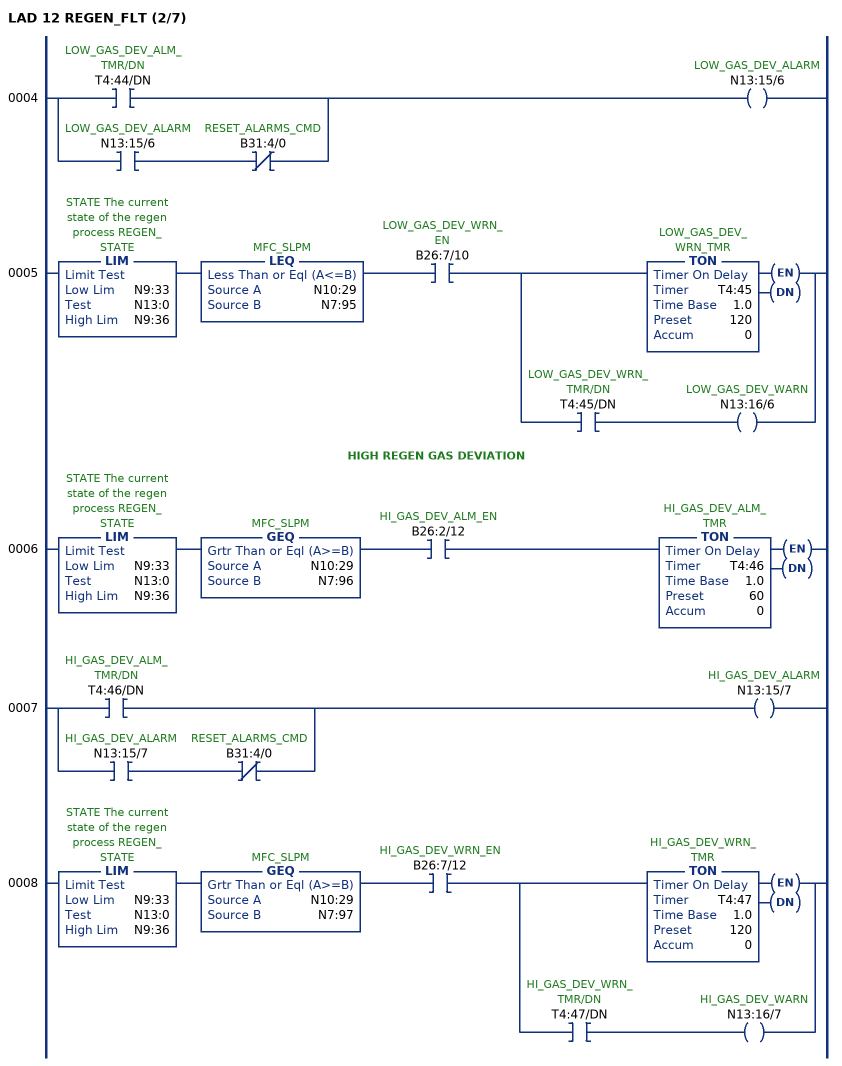
% Rung: 4 %
SOR BST XIC T4:44/DN NXB XIC N13:15/6 XIO B31:4/0 BND OTE N13:15/6 EOR
%   T4:44  LOW_GAS_DEV_ALM_TMR %
%   N13:15/6  LOW_GAS_DEV_ALARM %
%   B31:4/0  RESET_ALARMS_CMD %
% Rung: 5 %
SOR LIM N9:33 N13:0 N9:36 LEQ N10:29 N7:95 XIC B26:7/10 BST TON T4:45 1.0 120 0 NXB XIC T4:45/DN OTE N13:16/6 BND EOR
%   N9:33  REGEN_HEAT_BED  "STATE Regen Heat wall" %
%   N13:0  REGEN_STATE  "STATE The current state of the regen process" %
%   N9:36  REGEN_COOL  "STATE Regen Cool" %
%   N10:29  MFC_SLPM %
%   N7:95  LOW_GAS_DEV_WRN_SP %
%   B26:7/10  LOW_GAS_DEV_WRN_EN %
%   T4:45  LOW_GAS_DEV_WRN_TMR %
%   N13:16/6  LOW_GAS_DEV_WARN %
% Rung: 6 %
% TITLE: HIGH REGEN GAS DEVIATION %
SOR LIM N9:33 N13:0 N9:36 GEQ N10:29 N7:96 XIC B26:2/12 TON T4:46 1.0 60 0 EOR
%   N9:33  REGEN_HEAT_BED  "STATE Regen Heat wall" %
%   N13:0  REGEN_STATE  "STATE The current state of the regen process" %
%   N9:36  REGEN_COOL  "STATE Regen Cool" %
%   N10:29  MFC_SLPM %
%   N7:96  HI_GAS_DEV_ALM_SP %
%   B26:2/12  HI_GAS_DEV_ALM_EN %
%   T4:46  HI_GAS_DEV_ALM_TMR %
% Rung: 7 %
SOR BST XIC T4:46/DN NXB XIC N13:15/7 XIO B31:4/0 BND OTE N13:15/7 EOR
%   T4:46  HI_GAS_DEV_ALM_TMR %
%   N13:15/7  HI_GAS_DEV_ALARM %
%   B31:4/0  RESET_ALARMS_CMD %
% Rung: 8 %
SOR LIM N9:33 N13:0 N9:36 GEQ N10:29 N7:97 XIC B26:7/12 BST TON T4:47 1.0 120 0 NXB XIC T4:47/DN OTE N13:16/7 BND EOR
%   N9:33  REGEN_HEAT_BED  "STATE Regen Heat wall" %
%   N13:0  REGEN_STATE  "STATE The current state of the regen process" %
%   N9:36  REGEN_COOL  "STATE Regen Cool" %
%   N10:29  MFC_SLPM %
%   N7:97  HI_GAS_DEV_WRN_SP %
%   B26:7/12  HI_GAS_DEV_WRN_EN %
%   T4:47  HI_GAS_DEV_WRN_TMR %
%   N13:16/7  HI_GAS_DEV_WARN %

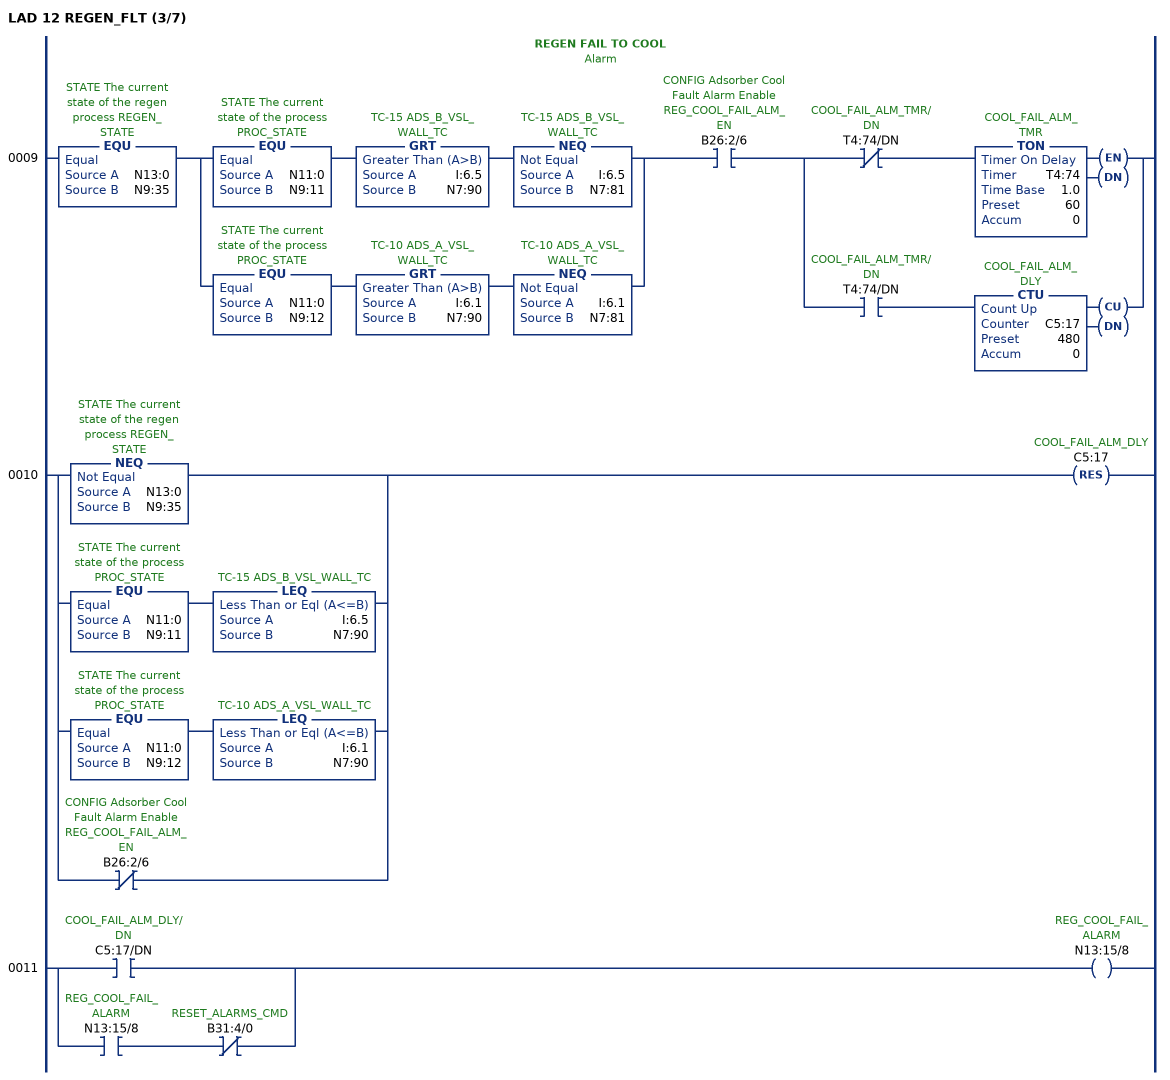
% Rung: 9 %
% TITLE: REGEN FAIL TO COOL %
% Alarm %
SOR EQU N13:0 N9:35 BST EQU N11:0 N9:11 GRT I:6.5 N7:90 NEQ I:6.5 N7:81 NXB EQU N11:0 N9:12 GRT I:6.1 N7:90 NEQ I:6.1 N7:81 BND XIC B26:2/6 BST XIO T4:74/DN TON T4:74 1.0 60 0 NXB XIC T4:74/DN CTU C5:17 480 0 BND EOR
%   N13:0  REGEN_STATE  "STATE The current state of the regen process" %
%   N9:35  REGEN_COOL_WALL  "STATE Regen Cool wall" %
%   N11:0  PROC_STATE  "STATE The current state of the process" %
%   N9:11  PROC_PFY_A_REG_B  "STATE Process Purify A" %
%   I:6.5  ADS_B_VSL_WALL_TC  "TC-15" %
%   N7:90  REG_COOL_FAIL_ALM_SP %
%   N7:81  TC_OPEN_SP  "CONFIG The value read by an open TC input" %
%   N9:12  PROC_PFY_B_REG_A  "STATE Process Purify B" %
%   I:6.1  ADS_A_VSL_WALL_TC  "TC-10" %
%   B26:2/6  REG_COOL_FAIL_ALM_EN  "CONFIG Adsorber Cool Fault Alarm Enable" %
%   T4:74  COOL_FAIL_ALM_TMR %
%   C5:17  COOL_FAIL_ALM_DLY %
% Rung: 10 %
SOR BST NEQ N13:0 N9:35 NXB EQU N11:0 N9:11 LEQ I:6.5 N7:90 NXB EQU N11:0 N9:12 LEQ I:6.1 N7:90 NXB XIO B26:2/6 BND RES C5:17 EOR
%   N13:0  REGEN_STATE  "STATE The current state of the regen process" %
%   N9:35  REGEN_COOL_WALL  "STATE Regen Cool wall" %
%   N11:0  PROC_STATE  "STATE The current state of the process" %
%   N9:11  PROC_PFY_A_REG_B  "STATE Process Purify A" %
%   I:6.5  ADS_B_VSL_WALL_TC  "TC-15" %
%   N7:90  REG_COOL_FAIL_ALM_SP %
%   N9:12  PROC_PFY_B_REG_A  "STATE Process Purify B" %
%   I:6.1  ADS_A_VSL_WALL_TC  "TC-10" %
%   B26:2/6  REG_COOL_FAIL_ALM_EN  "CONFIG Adsorber Cool Fault Alarm Enable" %
%   C5:17  COOL_FAIL_ALM_DLY %
% Rung: 11 %
SOR BST XIC C5:17/DN NXB XIC N13:15/8 XIO B31:4/0 BND OTE N13:15/8 EOR
%   C5:17  COOL_FAIL_ALM_DLY %
%   N13:15/8  REG_COOL_FAIL_ALARM %
%   B31:4/0  RESET_ALARMS_CMD %

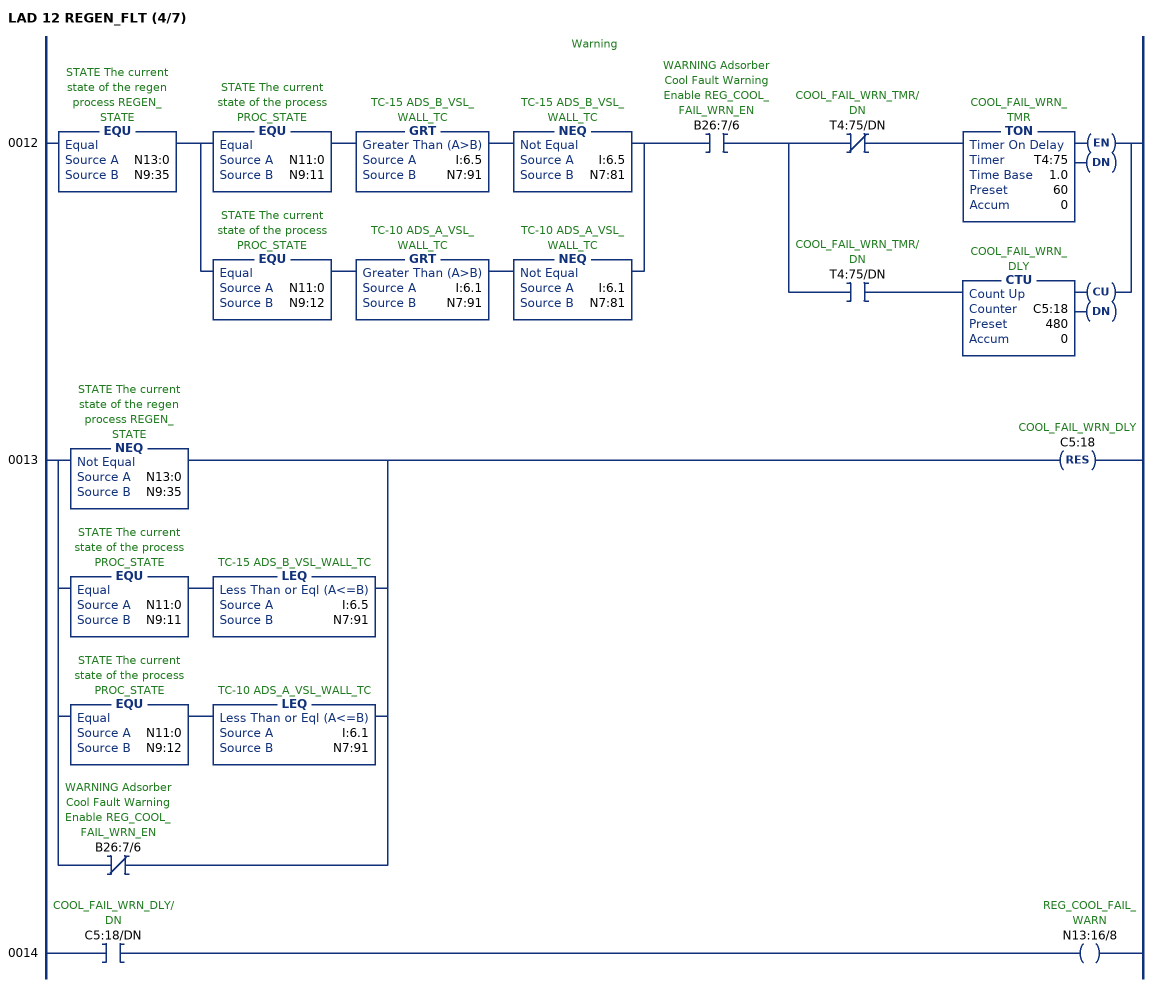
% Rung: 12 %
% Warning %
SOR EQU N13:0 N9:35 BST EQU N11:0 N9:11 GRT I:6.5 N7:91 NEQ I:6.5 N7:81 NXB EQU N11:0 N9:12 GRT I:6.1 N7:91 NEQ I:6.1 N7:81 BND XIC B26:7/6 BST XIO T4:75/DN TON T4:75 1.0 60 0 NXB XIC T4:75/DN CTU C5:18 480 0 BND EOR
%   N13:0  REGEN_STATE  "STATE The current state of the regen process" %
%   N9:35  REGEN_COOL_WALL  "STATE Regen Cool wall" %
%   N11:0  PROC_STATE  "STATE The current state of the process" %
%   N9:11  PROC_PFY_A_REG_B  "STATE Process Purify A" %
%   I:6.5  ADS_B_VSL_WALL_TC  "TC-15" %
%   N7:91  REG_COOL_FAIL_WRN_SP %
%   N7:81  TC_OPEN_SP  "CONFIG The value read by an open TC input" %
%   N9:12  PROC_PFY_B_REG_A  "STATE Process Purify B" %
%   I:6.1  ADS_A_VSL_WALL_TC  "TC-10" %
%   B26:7/6  REG_COOL_FAIL_WRN_EN  "WARNING Adsorber Cool Fault Warning Enable" %
%   T4:75  COOL_FAIL_WRN_TMR %
%   C5:18  COOL_FAIL_WRN_DLY %
% Rung: 13 %
SOR BST NEQ N13:0 N9:35 NXB EQU N11:0 N9:11 LEQ I:6.5 N7:91 NXB EQU N11:0 N9:12 LEQ I:6.1 N7:91 NXB XIO B26:7/6 BND RES C5:18 EOR
%   N13:0  REGEN_STATE  "STATE The current state of the regen process" %
%   N9:35  REGEN_COOL_WALL  "STATE Regen Cool wall" %
%   N11:0  PROC_STATE  "STATE The current state of the process" %
%   N9:11  PROC_PFY_A_REG_B  "STATE Process Purify A" %
%   I:6.5  ADS_B_VSL_WALL_TC  "TC-15" %
%   N7:91  REG_COOL_FAIL_WRN_SP %
%   N9:12  PROC_PFY_B_REG_A  "STATE Process Purify B" %
%   I:6.1  ADS_A_VSL_WALL_TC  "TC-10" %
%   B26:7/6  REG_COOL_FAIL_WRN_EN  "WARNING Adsorber Cool Fault Warning Enable" %
%   C5:18  COOL_FAIL_WRN_DLY %
% Rung: 14 %
SOR XIC C5:18/DN OTE N13:16/8 EOR
%   C5:18  COOL_FAIL_WRN_DLY %
%   N13:16/8  REG_COOL_FAIL_WARN %

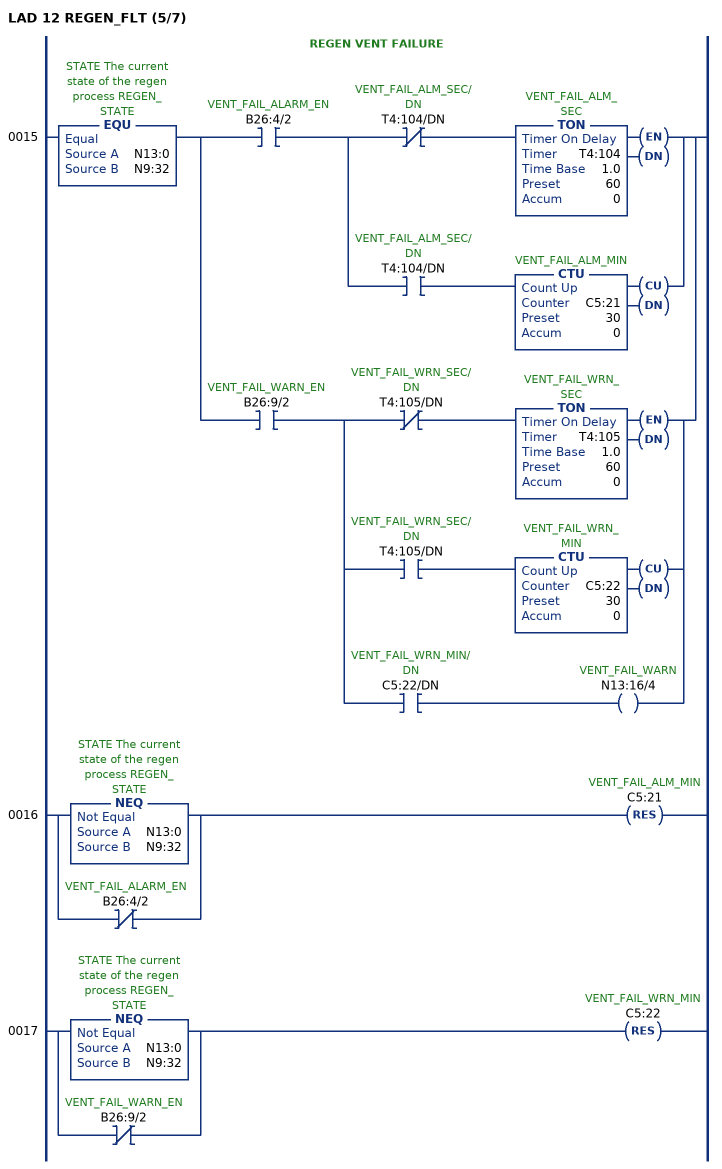
% Rung: 15 %
% TITLE: REGEN VENT FAILURE %
SOR EQU N13:0 N9:32 BST XIC B26:4/2 BST XIO T4:104/DN TON T4:104 1.0 60 0 NXB XIC T4:104/DN CTU C5:21 30 0 BND NXB XIC B26:9/2 BST XIO T4:105/DN TON T4:105 1.0 60 0 NXB XIC T4:105/DN CTU C5:22 30 0 NXB XIC C5:22/DN OTE N13:16/4 BND BND EOR
%   N13:0  REGEN_STATE  "STATE The current state of the regen process" %
%   N9:32  REGEN_VENT  "STATE Regen Vent" %
%   B26:4/2  VENT_FAIL_ALARM_EN %
%   T4:104  VENT_FAIL_ALM_SEC %
%   C5:21  VENT_FAIL_ALM_MIN %
%   B26:9/2  VENT_FAIL_WARN_EN %
%   T4:105  VENT_FAIL_WRN_SEC %
%   C5:22  VENT_FAIL_WRN_MIN %
%   N13:16/4  VENT_FAIL_WARN %
% Rung: 16 %
SOR BST NEQ N13:0 N9:32 NXB XIO B26:4/2 BND RES C5:21 EOR
%   N13:0  REGEN_STATE  "STATE The current state of the regen process" %
%   N9:32  REGEN_VENT  "STATE Regen Vent" %
%   B26:4/2  VENT_FAIL_ALARM_EN %
%   C5:21  VENT_FAIL_ALM_MIN %
% Rung: 17 %
SOR BST NEQ N13:0 N9:32 NXB XIO B26:9/2 BND RES C5:22 EOR
%   N13:0  REGEN_STATE  "STATE The current state of the regen process" %
%   N9:32  REGEN_VENT  "STATE Regen Vent" %
%   B26:9/2  VENT_FAIL_WARN_EN %
%   C5:22  VENT_FAIL_WRN_MIN %

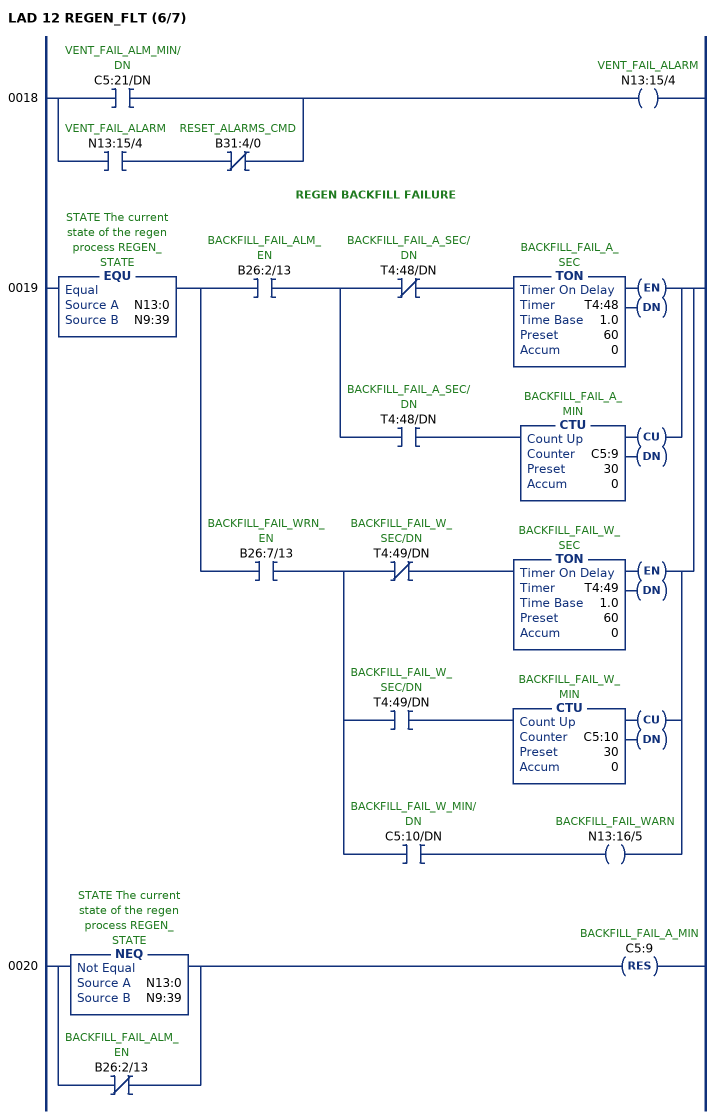
% Rung: 18 %
SOR BST XIC C5:21/DN NXB XIC N13:15/4 XIO B31:4/0 BND OTE N13:15/4 EOR
%   C5:21  VENT_FAIL_ALM_MIN %
%   N13:15/4  VENT_FAIL_ALARM %
%   B31:4/0  RESET_ALARMS_CMD %
% Rung: 19 %
% TITLE: REGEN BACKFILL FAILURE %
SOR EQU N13:0 N9:39 BST XIC B26:2/13 BST XIO T4:48/DN TON T4:48 1.0 60 0 NXB XIC T4:48/DN CTU C5:9 30 0 BND NXB XIC B26:7/13 BST XIO T4:49/DN TON T4:49 1.0 60 0 NXB XIC T4:49/DN CTU C5:10 30 0 NXB XIC C5:10/DN OTE N13:16/5 BND BND EOR
%   N13:0  REGEN_STATE  "STATE The current state of the regen process" %
%   N9:39  REGEN_BACKFILL %
%   B26:2/13  BACKFILL_FAIL_ALM_EN %
%   T4:48  BACKFILL_FAIL_A_SEC %
%   C5:9  BACKFILL_FAIL_A_MIN %
%   B26:7/13  BACKFILL_FAIL_WRN_EN %
%   T4:49  BACKFILL_FAIL_W_SEC %
%   C5:10  BACKFILL_FAIL_W_MIN %
%   N13:16/5  BACKFILL_FAIL_WARN %
% Rung: 20 %
SOR BST NEQ N13:0 N9:39 NXB XIO B26:2/13 BND RES C5:9 EOR
%   N13:0  REGEN_STATE  "STATE The current state of the regen process" %
%   N9:39  REGEN_BACKFILL %
%   B26:2/13  BACKFILL_FAIL_ALM_EN %
%   C5:9  BACKFILL_FAIL_A_MIN %

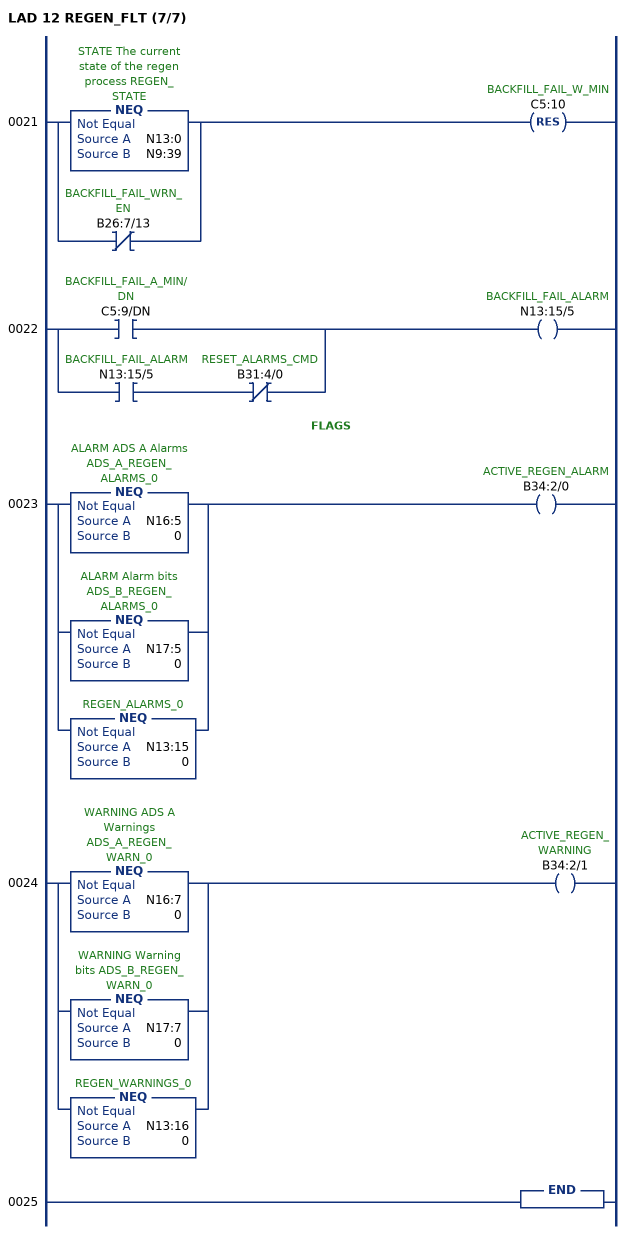
% Rung: 21 %
SOR BST NEQ N13:0 N9:39 NXB XIO B26:7/13 BND RES C5:10 EOR
%   N13:0  REGEN_STATE  "STATE The current state of the regen process" %
%   N9:39  REGEN_BACKFILL %
%   B26:7/13  BACKFILL_FAIL_WRN_EN %
%   C5:10  BACKFILL_FAIL_W_MIN %
% Rung: 22 %
SOR BST XIC C5:9/DN NXB XIC N13:15/5 XIO B31:4/0 BND OTE N13:15/5 EOR
%   C5:9  BACKFILL_FAIL_A_MIN %
%   N13:15/5  BACKFILL_FAIL_ALARM %
%   B31:4/0  RESET_ALARMS_CMD %
% Rung: 23 %
% TITLE: FLAGS %
SOR BST NEQ N16:5 0 NXB NEQ N17:5 0 NXB NEQ N13:15 0 BND OTE B34:2/0 EOR
%   N16:5  ADS_A_REGEN_ALARMS_0  "ALARM ADS A Alarms" %
%   N17:5  ADS_B_REGEN_ALARMS_0  "ALARM Alarm bits" %
%   N13:15  REGEN_ALARMS_0 %
%   B34:2/0  ACTIVE_REGEN_ALARM %
% Rung: 24 %
SOR BST NEQ N16:7 0 NXB NEQ N17:7 0 NXB NEQ N13:16 0 BND OTE B34:2/1 EOR
%   N16:7  ADS_A_REGEN_WARN_0  "WARNING ADS A Warnings" %
%   N17:7  ADS_B_REGEN_WARN_0  "WARNING Warning bits" %
%   N13:16  REGEN_WARNINGS_0 %
%   B34:2/1  ACTIVE_REGEN_WARNING %
% Rung: 25 %
SOR END EOR

LADDER 13 "PURGE"
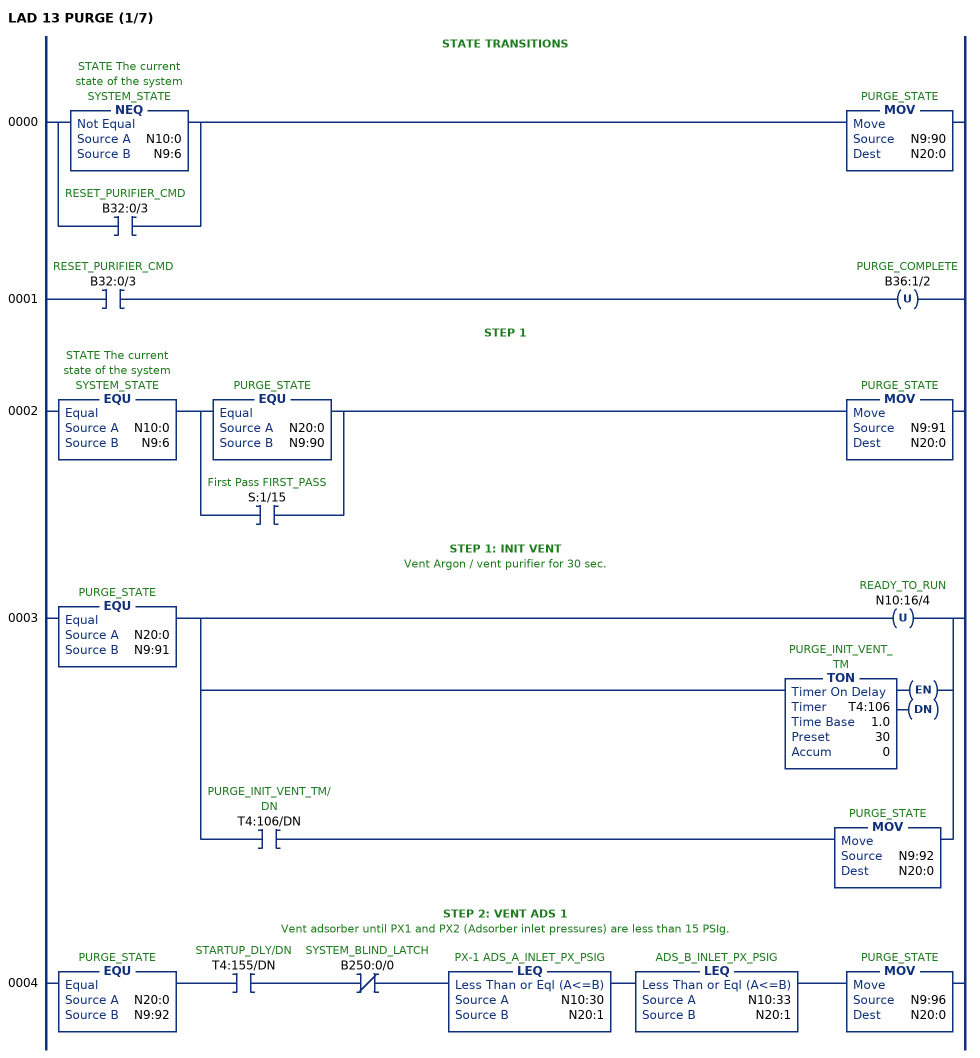
% Rung: 0 %
% TITLE: STATE TRANSITIONS %
SOR BST NEQ N10:0 N9:6 NXB XIC B32:0/3 BND MOV N9:90 N20:0 EOR
%   N10:0  SYSTEM_STATE  "STATE The current state of the system" %
%   N9:6  SYSTEM_PURGE %
%   B32:0/3  RESET_PURIFIER_CMD %
%   N9:90  PURGE_IDLE %
%   N20:0  PURGE_STATE %
% Rung: 1 %
SOR XIC B32:0/3 OTU B36:1/2 EOR
%   B32:0/3  RESET_PURIFIER_CMD %
%   B36:1/2  PURGE_COMPLETE %
% Rung: 2 %
% TITLE: STEP 1 %
SOR EQU N10:0 N9:6 BST EQU N20:0 N9:90 NXB XIC S:1/15 BND MOV N9:91 N20:0 EOR
%   N10:0  SYSTEM_STATE  "STATE The current state of the system" %
%   N9:6  SYSTEM_PURGE %
%   N20:0  PURGE_STATE %
%   N9:90  PURGE_IDLE %
%   S:1/15  FIRST_PASS  "First Pass" %
%   N9:91  PURGE_INIT_VENT %
% Rung: 3 %
% TITLE: STEP 1: INIT VENT %
% Vent Argon / vent purifier for 30 sec. %
SOR EQU N20:0 N9:91 BST OTU N10:16/4 NXB TON T4:106 1.0 30 0 NXB XIC T4:106/DN MOV N9:92 N20:0 BND EOR
%   N20:0  PURGE_STATE %
%   N9:91  PURGE_INIT_VENT %
%   N10:16/4  READY_TO_RUN %
%   T4:106  PURGE_INIT_VENT_TM %
%   N9:92  PURGE_VENT_ADSORBER %
% Rung: 4 %
% TITLE: STEP 2: VENT ADS 1 %
% Vent adsorber until PX1 and PX2 (Adsorber inlet pressures) are less than 15 PSIg. %
SOR EQU N20:0 N9:92 XIC T4:155/DN XIO B250:0/0 LEQ N10:30 N20:1 LEQ N10:33 N20:1 MOV N9:96 N20:0 EOR
%   N20:0  PURGE_STATE %
%   N9:92  PURGE_VENT_ADSORBER %
%   T4:155  STARTUP_DLY %
%   B250:0/0  SYSTEM_BLIND_LATCH %
%   N10:30  ADS_A_INLET_PX_PSIG  "PX-1" %
%   N20:1  PURGE_VENT_ADS_PRES %
%   N10:33  ADS_B_INLET_PX_PSIG %
%   N9:96  PURGE_VENT_GETTER %

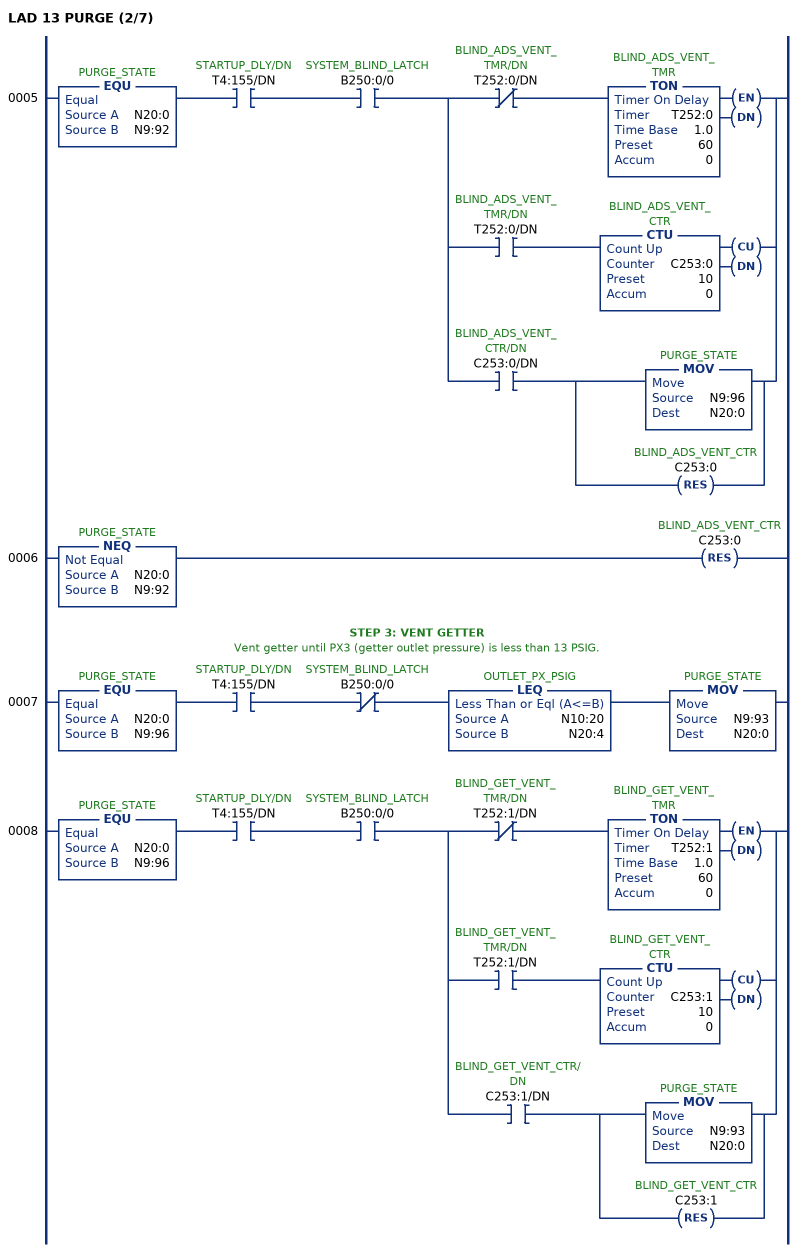
% Rung: 5 %
SOR EQU N20:0 N9:92 XIC T4:155/DN XIC B250:0/0 BST XIO T252:0/DN TON T252:0 1.0 60 0 NXB XIC T252:0/DN CTU C253:0 10 0 NXB XIC C253:0/DN BST MOV N9:96 N20:0 NXB RES C253:0 BND BND EOR
%   N20:0  PURGE_STATE %
%   N9:92  PURGE_VENT_ADSORBER %
%   T4:155  STARTUP_DLY %
%   B250:0/0  SYSTEM_BLIND_LATCH %
%   T252:0  BLIND_ADS_VENT_TMR %
%   C253:0  BLIND_ADS_VENT_CTR %
%   N9:96  PURGE_VENT_GETTER %
% Rung: 6 %
SOR NEQ N20:0 N9:92 RES C253:0 EOR
%   N20:0  PURGE_STATE %
%   N9:92  PURGE_VENT_ADSORBER %
%   C253:0  BLIND_ADS_VENT_CTR %
% Rung: 7 %
% TITLE: STEP 3: VENT GETTER %
% Vent getter until PX3 (getter outlet pressure) is less than 13 PSIG. %
SOR EQU N20:0 N9:96 XIC T4:155/DN XIO B250:0/0 LEQ N10:20 N20:4 MOV N9:93 N20:0 EOR
%   N20:0  PURGE_STATE %
%   N9:96  PURGE_VENT_GETTER %
%   T4:155  STARTUP_DLY %
%   B250:0/0  SYSTEM_BLIND_LATCH %
%   N10:20  OUTLET_PX_PSIG %
%   N20:4  PURGE_VENT_GET_PRES %
%   N9:93  PURGE_BACKFILL %
% Rung: 8 %
SOR EQU N20:0 N9:96 XIC T4:155/DN XIC B250:0/0 BST XIO T252:1/DN TON T252:1 1.0 60 0 NXB XIC T252:1/DN CTU C253:1 10 0 NXB XIC C253:1/DN BST MOV N9:93 N20:0 NXB RES C253:1 BND BND EOR
%   N20:0  PURGE_STATE %
%   N9:96  PURGE_VENT_GETTER %
%   T4:155  STARTUP_DLY %
%   B250:0/0  SYSTEM_BLIND_LATCH %
%   T252:1  BLIND_GET_VENT_TMR %
%   C253:1  BLIND_GET_VENT_CTR %
%   N9:93  PURGE_BACKFILL %

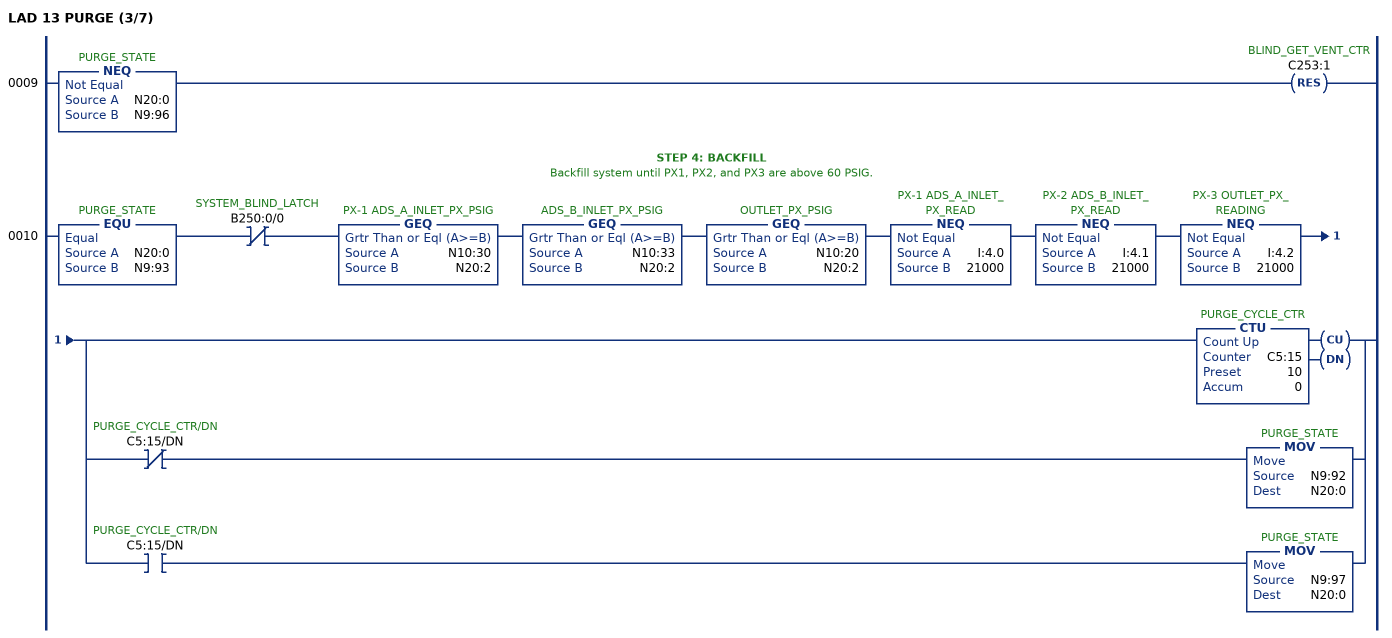
% Rung: 9 %
SOR NEQ N20:0 N9:96 RES C253:1 EOR
%   N20:0  PURGE_STATE %
%   N9:96  PURGE_VENT_GETTER %
%   C253:1  BLIND_GET_VENT_CTR %
% Rung: 10 %
% TITLE: STEP 4: BACKFILL %
% Backfill system until PX1, PX2, and PX3 are above 60 PSIG. %
SOR EQU N20:0 N9:93 XIO B250:0/0 GEQ N10:30 N20:2 GEQ N10:33 N20:2 GEQ N10:20 N20:2 NEQ I:4.0 21000 NEQ I:4.1 21000 NEQ I:4.2 21000 BST CTU C5:15 10 0 NXB XIO C5:15/DN MOV N9:92 N20:0 NXB XIC C5:15/DN MOV N9:97 N20:0 BND EOR
%   N20:0  PURGE_STATE %
%   N9:93  PURGE_BACKFILL %
%   B250:0/0  SYSTEM_BLIND_LATCH %
%   N10:30  ADS_A_INLET_PX_PSIG  "PX-1" %
%   N20:2  PURGE_BKFIL_PRES %
%   N10:33  ADS_B_INLET_PX_PSIG %
%   N10:20  OUTLET_PX_PSIG %
%   I:4.0  ADS_A_INLET_PX_READ  "PX-1" %
%   I:4.1  ADS_B_INLET_PX_READ  "PX-2" %
%   I:4.2  OUTLET_PX_READING  "PX-3" %
%   C5:15  PURGE_CYCLE_CTR %
%   N9:92  PURGE_VENT_ADSORBER %
%   N9:97  PURGE_VENT_ADS_2 %

